LIN {X 0,Y 367.075,Z 1146.88,A -85,B 0,C 180,E1 14634.153,E2 14634.153} C_VEL
LIN {X 0,Y 373.267,Z 1130.589,A -85,B 0,C 180,E1 14631.284,E2 14631.284} C_VEL
LIN {X 0,Y 379.59,Z 1113.754,A -85,B 0,C 180,E1 14628.758,E2 14628.758} C_VEL
LIN {X 0,Y 386.074,Z 1095.539,A -85,B 0,C 180,E1 14626.458,E2 14626.458} C_VEL
LIN {X 0,Y 392.313,Z 1077.12,A -85,B 0,C 180,E1 14624.47,E2 14624.47} C_VEL
LIN {X 0,Y 398.602,Z 1056.8,A -85,B 0,C 180,E1 14622.633,E2 14622.633} C_VEL
LIN {X 0,Y 404.177,Z 1037.14,A -85,B 0,C 180,E1 14621.125,E2 14621.125} C_VEL
LIN {X 0,Y 409.615,Z 1015.322,A -85,B 0,C 180,E1 14619.744,E2 14619.744} C_VEL
LIN {X 0,Y 414.222,Z 994.195,A -85,B 0,C 180,E1 14618.639,E2 14618.639} C_VEL
LIN {X 0,Y 418.394,Z 971.046,A -85,B 0,C 180,E1 14617.677,E2 14617.677} C_VEL
LIN {X 0,Y 421.612,Z 949.02,A -85,B 0,C 180,E1 14616.963,E2 14616.963} C_VEL
LIN {X 0,Y 424.148,Z 924.511,A -85,B 0,C 180,E1 14616.384,E2 14616.384} C_VEL
LIN {X 0,Y 439.358,Z 688.452,A -85,B 0,C 180,E1 14612.27,E2 14612.27} C_VEL
LIN {X 0,Y 440.922,Z 663.001,A -85,B 0,C 180,E1 14611.82,E2 14611.82} C_VEL
LIN {X 0,Y 431.754,Z 648.158,A -85,B 0,C 180,E1 14609.595,E2 14609.595} C_VEL
LIN {X 0,Y 422.609,Z 634.496,A -85,B 0,C 180,E1 14607.17,E2 14607.17} C_VEL
LIN {X 0,Y 413.735,Z 622.138,A -85,B 0,C 180,E1 14604.562,E2 14604.562} C_VEL
LIN {X 0,Y 405.049,Z 611.055,A -85,B 0,C 180,E1 14601.695,E2 14601.695} C_VEL
LIN {X 0,Y 397.899,Z 602.317,A -85,B 0,C 180,E1 14598.991,E2 14598.991} C_VEL
LIN {X 0,Y 392.596,Z 596.37,A -85,B 0,C 180,E1 14596.726,E2 14596.726} C_VEL
LIN {X 0,Y 388.549,Z 591.744,A -85,B 0,C 180,E1 14594.76,E2 14594.76} C_VEL
LIN {X 0,Y 383.66,Z 586.476,A -85,B 0,C 180,E1 14592.034,E2 14592.034} C_VEL
LIN {X 0,Y 379.03,Z 581.897,A -85,B 0,C 180,E1 14588.878,E2 14588.878} C_VEL
LIN {X 0,Y 378.199,Z 580.649,A -85,B 0,C 180,E1 14587.749,E2 14587.749} C_VEL
LIN {X 0,Y 376.427,Z 578.063,A -85,B 0,C 180,E1 14582.131,E2 14582.131} C_VEL
LIN {X 0,Y 376.328,Z 577.802,A -85,B 0,C 180,E1 14578.477,E2 14578.477} C_VEL
LIN {X 0,Y 377.214,Z 579.561,A -85,B 0,C 180,E1 14573.608,E2 14573.608} C_VEL
LIN {X 0,Y 378.457,Z 581.248,A -85,B 0,C 180,E1 14570.879,E2 14570.879} C_VEL
LIN {X 0,Y 380.862,Z 586.157,A -85,B 0,C 180,E1 14566.488,E2 14566.488} C_VEL
LIN {X 0,Y 383.165,Z 591.028,A -85,B 0,C 180,E1 14563.318,E2 14563.318} C_VEL
LIN {X 0,Y 385.362,Z 595.637,A -85,B 0,C 180,E1 14560.809,E2 14560.809} C_VEL
LIN {X 0,Y 387.472,Z 600.181,A -85,B 0,C 180,E1 14558.663,E2 14558.663} C_VEL
LIN {X 0,Y 389.455,Z 603.852,A -85,B 0,C 180,E1 14557.19,E2 14557.19} C_VEL
LIN {X 0,Y 396.46,Z 614.138,A -85,B 0,C 180,E1 14554.01,E2 14554.01} C_VEL
LIN {X 0,Y 403.343,Z 624.564,A -85,B 0,C 180,E1 14551.335,E2 14551.335} C_VEL
LIN {X 0,Y 411.127,Z 636.839,A -85,B 0,C 180,E1 14548.677,E2 14548.677} C_VEL
LIN {X 0,Y 418.492,Z 649.282,A -85,B 0,C 180,E1 14546.419,E2 14546.419} C_VEL
LIN {X 0,Y 427.201,Z 664.773,A -85,B 0,C 180,E1 14544.001,E2 14544.001} C_VEL
LIN {X 0,Y 430.356,Z 671.029,A -85,B 0,C 180,E1 14543.17,E2 14543.17} C_VEL
LIN {X 0,Y 435.237,Z 722.791,A -85,B 0,C 180,E1 14540.824,E2 14540.824} C_VEL
LIN {X 0,Y 423.088,Z 947.316,A -85,B 0,C 180,E1 14537.248,E2 14537.248} C_VEL
LIN {X 0,Y 420.542,Z 970.15,A -85,B 0,C 180,E1 14536.723,E2 14536.723} C_VEL
LIN {X 0,Y 417.124,Z 991.912,A -85,B 0,C 180,E1 14536.04,E2 14536.04} C_VEL
LIN {X 0,Y 413.008,Z 1012.312,A -85,B 0,C 180,E1 14535.18,E2 14535.18} C_VEL
LIN {X 0,Y 407.851,Z 1033.865,A -85,B 0,C 180,E1 14534.028,E2 14534.028} C_VEL
LIN {X 0,Y 402.694,Z 1052.364,A -85,B 0,C 180,E1 14532.803,E2 14532.803} C_VEL
LIN {X 0,Y 396.609,Z 1071.682,A -85,B 0,C 180,E1 14531.242,E2 14531.242} C_VEL
LIN {X 0,Y 390.215,Z 1090.083,A -85,B 0,C 180,E1 14529.454,E2 14529.454} C_VEL
LIN {X 0,Y 383.57,Z 1107.397,A -85,B 0,C 180,E1 14527.399,E2 14527.399} C_VEL
LIN {X 0,Y 376.663,Z 1124.336,A -85,B 0,C 180,E1 14524.986,E2 14524.986} C_VEL
LIN {X 0,Y 370.434,Z 1138.925,A -85,B 0,C 180,E1 14522.488,E2 14522.488} C_VEL
LIN {X 0,Y 364.569,Z 1152.135,A -85,B 0,C 180,E1 14519.762,E2 14519.762} C_VEL
LIN {X 0,Y 359.259,Z 1164.199,A -85,B 0,C 180,E1 14516.799,E2 14516.799} C_VEL
LIN {X 0,Y 354.544,Z 1174.916,A -85,B 0,C 180,E1 14513.569,E2 14513.569} C_VEL
LIN {X 0,Y 350.568,Z 1184.53,A -85,B 0,C 180,E1 14510.014,E2 14510.014} C_VEL
LIN {X 0,Y 347.654,Z 1192.408,A -85,B 0,C 180,E1 14506.371,E2 14506.371} C_VEL
LIN {X 0,Y 345.722,Z 1198.398,A -85,B 0,C 180,E1 14502.697,E2 14502.697} C_VEL
LIN {X 0,Y 344.593,Z 1203.015,A -85,B 0,C 180,E1 14498.846,E2 14498.846} C_VEL
LIN {X 0,Y 344.142,Z 1205.734,A -85,B 0,C 180,E1 14495.335,E2 14495.335} C_VEL
LIN {X 0,Y 344.006,Z 1207.141,A -85,B 0,C 180,E1 14491.666,E2 14491.666} C_VEL
LIN {X 0,Y 344,Z 1207.177,A -85,B 0,C 180,E1 14488.501,E2 14488.501} C_VEL
LIN {X 0,Y 344.124,Z 1205.916,A -85,B 0,C 180,E1 14484.832,E2 14484.832} C_VEL
LIN {X 0,Y 344.544,Z 1203.27,A -85,B 0,C 180,E1 14481.321,E2 14481.321} C_VEL
LIN {X 0,Y 345.693,Z 1198.563,A -85,B 0,C 180,E1 14477.302,E2 14477.302} C_VEL
LIN {X 0,Y 347.601,Z 1192.614,A -85,B 0,C 180,E1 14473.627,E2 14473.627} C_VEL
LIN {X 0,Y 350.493,Z 1184.79,A -85,B 0,C 180,E1 14469.981,E2 14469.981} C_VEL
LIN {X 0,Y 354.698,Z 1174.638,A -85,B 0,C 180,E1 14466.228,E2 14466.228} C_VEL
LIN {X 0,Y 359.396,Z 1164.003,A -85,B 0,C 180,E1 14463.033,E2 14463.033} C_VEL
LIN {X 0,Y 364.916,Z 1151.502,A -85,B 0,C 180,E1 14459.981,E2 14459.981} C_VEL
LIN {X 0,Y 371.322,Z 1136.991,A -85,B 0,C 180,E1 14457.049,E2 14457.049} C_VEL
LIN {X 0,Y 377.667,Z 1122.208,A -85,B 0,C 180,E1 14454.564,E2 14454.564} C_VEL
LIN {X 0,Y 384.244,Z 1105.923,A -85,B 0,C 180,E1 14452.302,E2 14452.302} C_VEL
LIN {X 0,Y 390.941,Z 1088.307,A -85,B 0,C 180,E1 14450.254,E2 14450.254} C_VEL
LIN {X 0,Y 396.895,Z 1071.164,A -85,B 0,C 180,E1 14448.602,E2 14448.602} C_VEL
LIN {X 0,Y 400.054,Z 1061.338,A -85,B 0,C 180,E1 14447.776,E2 14447.776} C_VEL
LIN {X 0,Y 401.438,Z 1054.915,A -85,B 0,C 180,E1 14447.179,E2 14447.179} C_VEL
LIN {X 0,Y 401.841,Z 1038.851,A -85,B 0,C 180,E1 14445.454,E2 14445.454} C_VEL
LIN {X 0,Y 402.944,Z 1032.138,A -85,B 0,C 180,E1 14444.927,E2 14444.927} C_VEL
LIN {X 0,Y 408.068,Z 1010.972,A -85,B 0,C 180,E1 14443.814,E2 14443.814} C_VEL
LIN {X 0,Y 412.471,Z 989.311,A -85,B 0,C 180,E1 14442.921,E2 14442.921} C_VEL
LIN {X 0,Y 415.872,Z 967.674,A -85,B 0,C 180,E1 14442.264,E2 14442.264} C_VEL
LIN {X 0,Y 418.4,Z 943.81,A -85,B 0,C 180,E1 14441.739,E2 14441.739} C_VEL
LIN {X 0,Y 430.607,Z 723.448,A -85,B 0,C 180,E1 14438.192,E2 14438.192} C_VEL
LIN {X 0,Y 426.313,Z 675.47,A -85,B 0,C 180,E1 14435.982,E2 14435.982} C_VEL
LIN {X 0,Y 418.355,Z 660.566,A -85,B 0,C 180,E1 14433.758,E2 14433.758} C_VEL
LIN {X 0,Y 410.661,Z 647.161,A -85,B 0,C 180,E1 14431.403,E2 14431.403} C_VEL
LIN {X 0,Y 402.691,Z 634.171,A -85,B 0,C 180,E1 14428.675,E2 14428.675} C_VEL
LIN {X 0,Y 397.146,Z 625.543,A -85,B 0,C 180,E1 14426.544,E2 14426.544} C_VEL
LIN {X 0,Y 391.843,Z 617.436,A -85,B 0,C 180,E1 14424.257,E2 14424.257} C_VEL
LIN {X 0,Y 386.128,Z 608.96,A -85,B 0,C 180,E1 14421.415,E2 14421.415} C_VEL
LIN {X 0,Y 380.176,Z 600.315,A -85,B 0,C 180,E1 14417.764,E2 14417.764} C_VEL
LIN {X 0,Y 377.816,Z 595.977,A -85,B 0,C 180,E1 14415.346,E2 14415.346} C_VEL
LIN {X 0,Y 375.944,Z 591.854,A -85,B 0,C 180,E1 14412.441,E2 14412.441} C_VEL
LIN {X 0,Y 373.797,Z 587.386,A -85,B 0,C 180,E1 14407.996,E2 14407.996} C_VEL
LIN {X 0,Y 372.205,Z 585.048,A -85,B 0,C 180,E1 14402.463,E2 14402.463} C_VEL
LIN {X 0,Y 372.164,Z 584.871,A -85,B 0,C 180,E1 14398.922,E2 14398.922} C_VEL
LIN {X 0,Y 372.818,Z 585.725,A -85,B 0,C 180,E1 14396.617,E2 14396.617} C_VEL
LIN {X 0,Y 377.49,Z 589.328,A -85,B 0,C 180,E1 14391.777,E2 14391.777} C_VEL
LIN {X 0,Y 381.514,Z 593.671,A -85,B 0,C 180,E1 14388.817,E2 14388.817} C_VEL
LIN {X 0,Y 383.391,Z 595.508,A -85,B 0,C 180,E1 14387.651,E2 14387.651} C_VEL
LIN {X 0,Y 388.761,Z 601.407,A -85,B 0,C 180,E1 14384.714,E2 14384.714} C_VEL
LIN {X 0,Y 394.144,Z 607.712,A -85,B 0,C 180,E1 14382.2,E2 14382.2} C_VEL
LIN {X 0,Y 398.695,Z 613.148,A -85,B 0,C 180,E1 14380.325,E2 14380.325} C_VEL
LIN {X 0,Y 405.06,Z 621.01,A -85,B 0,C 180,E1 14377.962,E2 14377.962} C_VEL
LIN {X 0,Y 414.608,Z 633.741,A -85,B 0,C 180,E1 14374.846,E2 14374.846} C_VEL
LIN {X 0,Y 423.799,Z 647.185,A -85,B 0,C 180,E1 14372.189,E2 14372.189} C_VEL
LIN {X 0,Y 433.257,Z 662.083,A -85,B 0,C 180,E1 14369.717,E2 14369.717} C_VEL
LIN {X 0,Y 436.289,Z 667.482,A -85,B 0,C 180,E1 14368.959,E2 14368.959} C_VEL
LIN {X 0,Y 420.331,Z 909.767,A -85,B 0,C 180,E1 14364.754,E2 14364.754} C_VEL
LIN {X 0,Y 417.975,Z 937.62,A -85,B 0,C 180,E1 14364.195,E2 14364.195} C_VEL
LIN {X 0,Y 414.977,Z 961.048,A -85,B 0,C 180,E1 14363.542,E2 14363.542} C_VEL
LIN {X 0,Y 411.076,Z 983.796,A -85,B 0,C 180,E1 14362.689,E2 14362.689} C_VEL
LIN {X 0,Y 406.363,Z 1006.888,A -85,B 0,C 180,E1 14361.598,E2 14361.598} C_VEL
LIN {X 0,Y 400.948,Z 1028.836,A -85,B 0,C 180,E1 14360.293,E2 14360.293} C_VEL
LIN {X 0,Y 394.958,Z 1050.407,A -85,B 0,C 180,E1 14358.753,E2 14358.753} C_VEL
LIN {X 0,Y 388.718,Z 1070.338,A -85,B 0,C 180,E1 14357.027,E2 14357.027} C_VEL
LIN {X 0,Y 381.72,Z 1090.963,A -85,B 0,C 180,E1 14354.903,E2 14354.903} C_VEL
LIN {X 0,Y 375.382,Z 1108.288,A -85,B 0,C 180,E1 14352.782,E2 14352.782} C_VEL
LIN {X 0,Y 368.175,Z 1127.067,A -85,B 0,C 180,E1 14350.062,E2 14350.062} C_VEL
LIN {X 0,Y 362.387,Z 1141.642,A -85,B 0,C 180,E1 14347.572,E2 14347.572} C_VEL
LIN {X 0,Y 355.922,Z 1157.783,A -85,B 0,C 180,E1 14344.316,E2 14344.316} C_VEL
LIN {X 0,Y 350.848,Z 1170.642,A -85,B 0,C 180,E1 14341.242,E2 14341.242} C_VEL
LIN {X 0,Y 345.924,Z 1183.598,A -85,B 0,C 180,E1 14337.546,E2 14337.546} C_VEL
LIN {X 0,Y 342.26,Z 1194.124,A -85,B 0,C 180,E1 14333.958,E2 14333.958} C_VEL
LIN {X 0,Y 339.449,Z 1203.219,A -85,B 0,C 180,E1 14330.159,E2 14330.159} C_VEL
LIN {X 0,Y 337.719,Z 1210.045,A -85,B 0,C 180,E1 14326.689,E2 14326.689} C_VEL
LIN {X 0,Y 336.509,Z 1216.429,A -85,B 0,C 180,E1 14322.527,E2 14322.527} C_VEL
LIN {X 0,Y 336.076,Z 1220.328,A -85,B 0,C 180,E1 14319.072,E2 14319.072} C_VEL
LIN {X 0,Y 335.938,Z 1223.253,A -85,B 0,C 180,E1 14315.294,E2 14315.294} C_VEL
LIN {X 0,Y 335.967,Z 1224.501,A -85,B 0,C 180,E1 14311.705,E2 14311.705} C_VEL
LIN {X 0,Y 335.969,Z 1224.547,A -85,B 0,C 180,E1 14308.636,E2 14308.636} C_VEL
LIN {X 0,Y 335.949,Z 1223.537,A -85,B 0,C 180,E1 14305.391,E2 14305.391} C_VEL
LIN {X 0,Y 336.03,Z 1220.984,A -85,B 0,C 180,E1 14301.616,E2 14301.616} C_VEL
LIN {X 0,Y 336.414,Z 1217.058,A -85,B 0,C 180,E1 14297.992,E2 14297.992} C_VEL
LIN {X 0,Y 337.33,Z 1211.819,A -85,B 0,C 180,E1 14294.352,E2 14294.352} C_VEL
LIN {X 0,Y 339.139,Z 1204.281,A -85,B 0,C 180,E1 14290.361,E2 14290.361} C_VEL
LIN {X 0,Y 341.68,Z 1195.859,A -85,B 0,C 180,E1 14286.731,E2 14286.731} C_VEL
LIN {X 0,Y 345.337,Z 1185.139,A -85,B 0,C 180,E1 14282.963,E2 14282.963} C_VEL
LIN {X 0,Y 349.618,Z 1173.731,A -85,B 0,C 180,E1 14279.589,E2 14279.589} C_VEL
LIN {X 0,Y 355.013,Z 1159.928,A -85,B 0,C 180,E1 14276.188,E2 14276.188} C_VEL
LIN {X 0,Y 361.027,Z 1144.988,A -85,B 0,C 180,E1 14273.06,E2 14273.06} C_VEL
LIN {X 0,Y 367.396,Z 1128.826,A -85,B 0,C 180,E1 14270.242,E2 14270.242} C_VEL
LIN {X 0,Y 374.235,Z 1111.205,A -85,B 0,C 180,E1 14267.621,E2 14267.621} C_VEL
LIN {X 0,Y 380.574,Z 1093.875,A -85,B 0,C 180,E1 14265.455,E2 14265.455} C_VEL
LIN {X 0,Y 387.377,Z 1074.25,A -85,B 0,C 180,E1 14263.361,E2 14263.361} C_VEL
LIN {X 0,Y 393.417,Z 1055.087,A -85,B 0,C 180,E1 14261.652,E2 14261.652} C_VEL
LIN {X 0,Y 399.608,Z 1033.598,A -85,B 0,C 180,E1 14260.036,E2 14260.036} C_VEL
LIN {X 0,Y 404.692,Z 1013.376,A -85,B 0,C 180,E1 14258.786,E2 14258.786} C_VEL
LIN {X 0,Y 409.537,Z 991.477,A -85,B 0,C 180,E1 14257.662,E2 14257.662} C_VEL
LIN {X 0,Y 413.522,Z 969.319,A -85,B 0,C 180,E1 14256.767,E2 14256.767} C_VEL
LIN {X 0,Y 416.916,Z 946.2,A -85,B 0,C 180,E1 14256.036,E2 14256.036} C_VEL
LIN {X 0,Y 419.267,Z 922.548,A -85,B 0,C 180,E1 14255.498,E2 14255.498} C_VEL
LIN {X 0,Y 435.003,Z 684.514,A -85,B 0,C 180,E1 14251.344,E2 14251.344} C_VEL
LIN {X 0,Y 436.072,Z 666.851,A -85,B 0,C 180,E1 14251.02,E2 14251.02} C_VEL
LIN {X 0,Y 426.546,Z 651.468,A -85,B 0,C 180,E1 14248.607,E2 14248.607} C_VEL
LIN {X 0,Y 417.357,Z 637.74,A -85,B 0,C 180,E1 14246.042,E2 14246.042} C_VEL
LIN {X 0,Y 408.027,Z 624.866,A -85,B 0,C 180,E1 14243.123,E2 14243.123} C_VEL
LIN {X 0,Y 399.618,Z 614.248,A -85,B 0,C 180,E1 14240.123,E2 14240.123} C_VEL
LIN {X 0,Y 394.405,Z 608.036,A -85,B 0,C 180,E1 14238.017,E2 14238.017} C_VEL
LIN {X 0,Y 390.537,Z 603.573,A -85,B 0,C 180,E1 14236.281,E2 14236.281} C_VEL
LIN {X 0,Y 386.859,Z 599.291,A -85,B 0,C 180,E1 14234.443,E2 14234.443} C_VEL
LIN {X 0,Y 382.19,Z 594.174,A -85,B 0,C 180,E1 14231.775,E2 14231.775} C_VEL
LIN {X 0,Y 377.662,Z 589.568,A -85,B 0,C 180,E1 14228.603,E2 14228.603} C_VEL
LIN {X 0,Y 376.14,Z 588.195,A -85,B 0,C 180,E1 14227.331,E2 14227.331} C_VEL
LIN {X 0,Y 372.214,Z 584.956,A -85,B 0,C 180,E1 14222.617,E2 14222.617} C_VEL
LIN {X 0,Y 371.979,Z 584.446,A -85,B 0,C 180,E1 14218.922,E2 14218.922} C_VEL
LIN {X 0,Y 372.563,Z 585.871,A -85,B 0,C 180,E1 14214.456,E2 14214.456} C_VEL
LIN {X 0,Y 374.026,Z 587.938,A -85,B 0,C 180,E1 14210.925,E2 14210.925} C_VEL
LIN {X 0,Y 376.302,Z 592.669,A -85,B 0,C 180,E1 14206.634,E2 14206.634} C_VEL
LIN {X 0,Y 378.573,Z 597.575,A -85,B 0,C 180,E1 14203.426,E2 14203.426} C_VEL
LIN {X 0,Y 381.302,Z 602.118,A -85,B 0,C 180,E1 14201.183,E2 14201.183} C_VEL
LIN {X 0,Y 387.44,Z 610.898,A -85,B 0,C 180,E1 14197.665,E2 14197.665} C_VEL
LIN {X 0,Y 394.439,Z 621.431,A -85,B 0,C 180,E1 14194.392,E2 14194.392} C_VEL
LIN {X 0,Y 401.014,Z 631.624,A -85,B 0,C 180,E1 14191.763,E2 14191.763} C_VEL
LIN {X 0,Y 408.466,Z 643.595,A -85,B 0,C 180,E1 14189.147,E2 14189.147} C_VEL
LIN {X 0,Y 415.589,Z 655.893,A -85,B 0,C 180,E1 14186.896,E2 14186.896} C_VEL
LIN {X 0,Y 424.048,Z 671.21,A -85,B 0,C 180,E1 14184.483,E2 14184.483} C_VEL
LIN {X 0,Y 426.192,Z 675.798,A -85,B 0,C 180,E1 14183.892,E2 14183.892} C_VEL
LIN {X 0,Y 430.502,Z 724.672,A -85,B 0,C 180,E1 14181.658,E2 14181.658} C_VEL
LIN {X 0,Y 418.035,Z 946.95,A -85,B 0,C 180,E1 14178.099,E2 14178.099} C_VEL
LIN {X 0,Y 415.411,Z 969.946,A -85,B 0,C 180,E1 14177.569,E2 14177.569} C_VEL
LIN {X 0,Y 411.915,Z 991.659,A -85,B 0,C 180,E1 14176.888,E2 14176.888} C_VEL
LIN {X 0,Y 407.724,Z 1011.938,A -85,B 0,C 180,E1 14176.034,E2 14176.034} C_VEL
LIN {X 0,Y 402.43,Z 1033.542,A -85,B 0,C 180,E1 14174.879,E2 14174.879} C_VEL
LIN {X 0,Y 396.9,Z 1052.853,A -85,B 0,C 180,E1 14173.594,E2 14173.594} C_VEL
LIN {X 0,Y 390.622,Z 1072.154,A -85,B 0,C 180,E1 14172.017,E2 14172.017} C_VEL
LIN {X 0,Y 384.048,Z 1090.491,A -85,B 0,C 180,E1 14170.215,E2 14170.215} C_VEL
LIN {X 0,Y 377.207,Z 1107.761,A -85,B 0,C 180,E1 14168.142,E2 14168.142} C_VEL
LIN {X 0,Y 370.077,Z 1124.648,A -85,B 0,C 180,E1 14165.703,E2 14165.703} C_VEL
LIN {X 0,Y 363.639,Z 1139.221,A -85,B 0,C 180,E1 14163.173,E2 14163.173} C_VEL
LIN {X 0,Y 357.558,Z 1152.397,A -85,B 0,C 180,E1 14160.407,E2 14160.407} C_VEL
LIN {X 0,Y 352.035,Z 1164.44,A -85,B 0,C 180,E1 14157.395,E2 14157.395} C_VEL
LIN {X 0,Y 347.164,Z 1175.045,A -85,B 0,C 180,E1 14154.14,E2 14154.14} C_VEL
LIN {X 0,Y 342.954,Z 1184.754,A -85,B 0,C 180,E1 14150.478,E2 14150.478} C_VEL
LIN {X 0,Y 339.886,Z 1192.626,A -85,B 0,C 180,E1 14146.756,E2 14146.756} C_VEL
LIN {X 0,Y 337.843,Z 1198.611,A -85,B 0,C 180,E1 14142.998,E2 14142.998} C_VEL
LIN {X 0,Y 336.639,Z 1203.222,A -85,B 0,C 180,E1 14139.057,E2 14139.057} C_VEL
LIN {X 0,Y 336.156,Z 1205.941,A -85,B 0,C 180,E1 14135.462,E2 14135.462} C_VEL
LIN {X 0,Y 336.009,Z 1207.345,A -85,B 0,C 180,E1 14131.705,E2 14131.705} C_VEL
LIN {X 0,Y 336.003,Z 1207.381,A -85,B 0,C 180,E1 14128.465,E2 14128.465} C_VEL
LIN {X 0,Y 336.136,Z 1206.122,A -85,B 0,C 180,E1 14124.709,E2 14124.709} C_VEL
LIN {X 0,Y 336.585,Z 1203.476,A -85,B 0,C 180,E1 14121.114,E2 14121.114} C_VEL
LIN {X 0,Y 337.812,Z 1198.774,A -85,B 0,C 180,E1 14117,E2 14117} C_VEL
LIN {X 0,Y 339.833,Z 1192.827,A -85,B 0,C 180,E1 14113.242,E2 14113.242} C_VEL
LIN {X 0,Y 342.877,Z 1185.011,A -85,B 0,C 180,E1 14109.517,E2 14109.517} C_VEL
LIN {X 0,Y 347.064,Z 1175.368,A -85,B 0,C 180,E1 14105.853,E2 14105.853} C_VEL
LIN {X 0,Y 351.911,Z 1164.797,A -85,B 0,C 180,E1 14102.595,E2 14102.595} C_VEL
LIN {X 0,Y 357.418,Z 1152.841,A -85,B 0,C 180,E1 14099.58,E2 14099.58} C_VEL
LIN {X 0,Y 363.832,Z 1138.95,A -85,B 0,C 180,E1 14096.664,E2 14096.664} C_VEL
LIN {X 0,Y 370.307,Z 1124.322,A -85,B 0,C 180,E1 14094.132,E2 14094.132} C_VEL
LIN {X 0,Y 377.464,Z 1107.365,A -85,B 0,C 180,E1 14091.696,E2 14091.696} C_VEL
LIN {X 0,Y 384.333,Z 1090.037,A -85,B 0,C 180,E1 14089.625,E2 14089.625} C_VEL
LIN {X 0,Y 390.92,Z 1071.626,A -85,B 0,C 180,E1 14087.825,E2 14087.825} C_VEL
LIN {X 0,Y 397.623,Z 1050.801,A -85,B 0,C 180,E1 14086.151,E2 14086.151} C_VEL
LIN {X 0,Y 402.944,Z 1032.138,A -85,B 0,C 180,E1 14084.927,E2 14084.927} C_VEL
LIN {X 0,Y 404.109,Z 1025.327,A -85,B 0,C 180,E1 14084.422,E2 14084.422} C_VEL
LIN {X 0,Y 404.184,Z 1008.202,A -85,B 0,C 180,E1 14082.925,E2 14082.925} C_VEL
LIN {X 0,Y 405.005,Z 1001.057,A -85,B 0,C 180,E1 14082.517,E2 14082.517} C_VEL
LIN {X 0,Y 408.853,Z 980.543,A -85,B 0,C 180,E1 14081.772,E2 14081.772} C_VEL
LIN {X 0,Y 412.137,Z 957.278,A -85,B 0,C 180,E1 14081.151,E2 14081.151} C_VEL
LIN {X 0,Y 414.107,Z 934.287,A -85,B 0,C 180,E1 14080.702,E2 14080.702} C_VEL
LIN {X 0,Y 425.986,Z 725.009,A -85,B 0,C 180,E1 14077.335,E2 14077.335} C_VEL
LIN {X 0,Y 422.146,Z 679.945,A -85,B 0,C 180,E1 14075.223,E2 14075.223} C_VEL
LIN {X 0,Y 414.286,Z 665.02,A -85,B 0,C 180,E1 14072.932,E2 14072.932} C_VEL
LIN {X 0,Y 406.152,Z 650.7,A -85,B 0,C 180,E1 14070.31,E2 14070.31} C_VEL
LIN {X 0,Y 398.248,Z 637.719,A -85,B 0,C 180,E1 14067.434,E2 14067.434} C_VEL
LIN {X 0,Y 390.354,Z 625.349,A -85,B 0,C 180,E1 14064.074,E2 14064.074} C_VEL
LIN {X 0,Y 384.379,Z 616.349,A -85,B 0,C 180,E1 14061.038,E2 14061.038} C_VEL
LIN {X 0,Y 378.669,Z 607.88,A -85,B 0,C 180,E1 14057.44,E2 14057.44} C_VEL
LIN {X 0,Y 375.726,Z 603.557,A -85,B 0,C 180,E1 14055.118,E2 14055.118} C_VEL
LIN {X 0,Y 372.866,Z 599.149,A -85,B 0,C 180,E1 14052.231,E2 14052.231} C_VEL
LIN {X 0,Y 370.187,Z 594.511,A -85,B 0,C 180,E1 14047.918,E2 14047.918} C_VEL
LIN {X 0,Y 369.372,Z 592.509,A -85,B 0,C 180,E1 14042.327,E2 14042.327} C_VEL
LIN {X 0,Y 370.667,Z 592.831,A -85,B 0,C 180,E1 14038.454,E2 14038.454} C_VEL
LIN {X 0,Y 373.543,Z 595.181,A -85,B 0,C 180,E1 14034.47,E2 14034.47} C_VEL
LIN {X 0,Y 376.227,Z 597.128,A -85,B 0,C 180,E1 14031.979,E2 14031.979} C_VEL
LIN {X 0,Y 380.298,Z 601.548,A -85,B 0,C 180,E1 14028.934,E2 14028.934} C_VEL
LIN {X 0,Y 382.028,Z 603.36,A -85,B 0,C 180,E1 14027.837,E2 14027.837} C_VEL
LIN {X 0,Y 387.191,Z 609.12,A -85,B 0,C 180,E1 14024.958,E2 14024.958} C_VEL
LIN {X 0,Y 392.341,Z 615.24,A -85,B 0,C 180,E1 14022.499,E2 14022.499} C_VEL
LIN {X 0,Y 398.203,Z 622.289,A -85,B 0,C 180,E1 14020.07,E2 14020.07} C_VEL
LIN {X 0,Y 406.204,Z 632.737,A -85,B 0,C 180,E1 14017.151,E2 14017.151} C_VEL
LIN {X 0,Y 415.104,Z 645.203,A -85,B 0,C 180,E1 14014.305,E2 14014.305} C_VEL
LIN {X 0,Y 424.045,Z 658.849,A -85,B 0,C 180,E1 14011.747,E2 14011.747} C_VEL
LIN {X 0,Y 431.56,Z 671.215,A -85,B 0,C 180,E1 14009.775,E2 14009.775} C_VEL
LIN {X 0,Y 415.043,Z 915.504,A -85,B 0,C 180,E1 14005.522,E2 14005.522} C_VEL
LIN {X 0,Y 412.777,Z 939.766,A -85,B 0,C 180,E1 14005.01,E2 14005.01} C_VEL
LIN {X 0,Y 409.536,Z 963.776,A -85,B 0,C 180,E1 14004.32,E2 14004.32} C_VEL
LIN {X 0,Y 405.599,Z 985.702,A -85,B 0,C 180,E1 14003.479,E2 14003.479} C_VEL
LIN {X 0,Y 400.746,Z 1008.459,A -85,B 0,C 180,E1 14002.381,E2 14002.381} C_VEL
LIN {X 0,Y 395.486,Z 1029.168,A -85,B 0,C 180,E1 14001.14,E2 14001.14} C_VEL
LIN {X 0,Y 389.325,Z 1050.692,A -85,B 0,C 180,E1 13999.593,E2 13999.593} C_VEL
LIN {X 0,Y 382.921,Z 1070.532,A -85,B 0,C 180,E1 13997.864,E2 13997.864} C_VEL
LIN {X 0,Y 375.678,Z 1091.182,A -85,B 0,C 180,E1 13995.72,E2 13995.72} C_VEL
LIN {X 0,Y 369.079,Z 1108.619,A -85,B 0,C 180,E1 13993.561,E2 13993.561} C_VEL
LIN {X 0,Y 361.473,Z 1127.69,A -85,B 0,C 180,E1 13990.752,E2 13990.752} C_VEL
LIN {X 0,Y 355.134,Z 1143.073,A -85,B 0,C 180,E1 13988.067,E2 13988.067} C_VEL
LIN {X 0,Y 348.789,Z 1158.21,A -85,B 0,C 180,E1 13984.926,E2 13984.926} C_VEL
LIN {X 0,Y 343.511,Z 1171.033,A -85,B 0,C 180,E1 13981.792,E2 13981.792} C_VEL
LIN {X 0,Y 338.583,Z 1183.352,A -85,B 0,C 180,E1 13978.196,E2 13978.196} C_VEL
LIN {X 0,Y 334.875,Z 1193.407,A -85,B 0,C 180,E1 13974.709,E2 13974.709} C_VEL
LIN {X 0,Y 331.724,Z 1202.993,A -85,B 0,C 180,E1 13970.65,E2 13970.65} C_VEL
LIN {X 0,Y 329.872,Z 1209.824,A -85,B 0,C 180,E1 13967.098,E2 13967.098} C_VEL
LIN {X 0,Y 328.569,Z 1216.217,A -85,B 0,C 180,E1 13962.835,E2 13962.835} C_VEL
LIN {X 0,Y 328.089,Z 1220.118,A -85,B 0,C 180,E1 13959.295,E2 13959.295} C_VEL
LIN {X 0,Y 327.941,Z 1223.047,A -85,B 0,C 180,E1 13955.423,E2 13955.423} C_VEL
LIN {X 0,Y 327.969,Z 1224.297,A -85,B 0,C 180,E1 13951.747,E2 13951.747} C_VEL
LIN {X 0,Y 327.972,Z 1224.342,A -85,B 0,C 180,E1 13948.602,E2 13948.602} C_VEL
LIN {X 0,Y 327.947,Z 1223.331,A -85,B 0,C 180,E1 13945.278,E2 13945.278} C_VEL
LIN {X 0,Y 328.049,Z 1220.773,A -85,B 0,C 180,E1 13941.411,E2 13941.411} C_VEL
LIN {X 0,Y 328.462,Z 1216.845,A -85,B 0,C 180,E1 13937.697,E2 13937.697} C_VEL
LIN {X 0,Y 329.523,Z 1211.334,A -85,B 0,C 180,E1 13933.79,E2 13933.79} C_VEL
LIN {X 0,Y 331.48,Z 1203.753,A -85,B 0,C 180,E1 13929.738,E2 13929.738} C_VEL
LIN {X 0,Y 334.395,Z 1194.772,A -85,B 0,C 180,E1 13925.818,E2 13925.818} C_VEL
LIN {X 0,Y 338.187,Z 1184.302,A -85,B 0,C 180,E1 13922.133,E2 13922.133} C_VEL
LIN {X 0,Y 342.991,Z 1172.258,A -85,B 0,C 180,E1 13918.547,E2 13918.547} C_VEL
LIN {X 0,Y 348.56,Z 1158.62,A -85,B 0,C 180,E1 13915.191,E2 13915.191} C_VEL
LIN {X 0,Y 354.768,Z 1143.811,A -85,B 0,C 180,E1 13912.092,E2 13912.092} C_VEL
LIN {X 0,Y 361.265,Z 1128.002,A -85,B 0,C 180,E1 13909.32,E2 13909.32} C_VEL
LIN {X 0,Y 368.465,Z 1110.005,A -85,B 0,C 180,E1 13906.644,E2 13906.644} C_VEL
LIN {X 0,Y 374.959,Z 1092.839,A -85,B 0,C 180,E1 13904.495,E2 13904.495} C_VEL
LIN {X 0,Y 382.157,Z 1072.52,A -85,B 0,C 180,E1 13902.344,E2 13902.344} C_VEL
LIN {X 0,Y 388.351,Z 1053.384,A -85,B 0,C 180,E1 13900.648,E2 13900.648} C_VEL
LIN {X 0,Y 394.913,Z 1030.858,A -85,B 0,C 180,E1 13898.988,E2 13898.988} C_VEL
LIN {X 0,Y 400.273,Z 1009.852,A -85,B 0,C 180,E1 13897.714,E2 13897.714} C_VEL
LIN {X 0,Y 405.282,Z 986.662,A -85,B 0,C 180,E1 13896.58,E2 13896.58} C_VEL
LIN {X 0,Y 409.25,Z 964.66,A -85,B 0,C 180,E1 13895.728,E2 13895.728} C_VEL
LIN {X 0,Y 412.577,Z 940.316,A -85,B 0,C 180,E1 13895.019,E2 13895.019} C_VEL
LIN {X 0,Y 414.858,Z 916.144,A -85,B 0,C 180,E1 13894.505,E2 13894.505} C_VEL
LIN {X 0,Y 431.263,Z 673.298,A -85,B 0,C 180,E1 13890.275,E2 13890.275} C_VEL
LIN {X 0,Y 431.29,Z 670.84,A -85,B 0,C 180,E1 13890.205,E2 13890.205} C_VEL
LIN {X 0,Y 422.219,Z 656.099,A -85,B 0,C 180,E1 13887.809,E2 13887.809} C_VEL
LIN {X 0,Y 414.094,Z 643.876,A -85,B 0,C 180,E1 13885.455,E2 13885.455} C_VEL
LIN {X 0,Y 405.546,Z 631.859,A -85,B 0,C 180,E1 13882.697,E2 13882.697} C_VEL
LIN {X 0,Y 397.558,Z 621.582,A -85,B 0,C 180,E1 13879.772,E2 13879.772} C_VEL
LIN {X 0,Y 392.439,Z 615.373,A -85,B 0,C 180,E1 13877.65,E2 13877.65} C_VEL
LIN {X 0,Y 388.212,Z 610.438,A -85,B 0,C 180,E1 13875.691,E2 13875.691} C_VEL
LIN {X 0,Y 385.182,Z 606.839,A -85,B 0,C 180,E1 13874.124,E2 13874.124} C_VEL
LIN {X 0,Y 380.729,Z 601.873,A -85,B 0,C 180,E1 13871.513,E2 13871.513} C_VEL
LIN {X 0,Y 376.216,Z 597.104,A -85,B 0,C 180,E1 13868.252,E2 13868.252} C_VEL
LIN {X 0,Y 370.891,Z 592.812,A -85,B 0,C 180,E1 13862.472,E2 13862.472} C_VEL
LIN {X 0,Y 369.23,Z 592.013,A -85,B 0,C 180,E1 13858.603,E2 13858.603} C_VEL
LIN {X 0,Y 369.278,Z 593.43,A -85,B 0,C 180,E1 13853.626,E2 13853.626} C_VEL
LIN {X 0,Y 370.256,Z 594.856,A -85,B 0,C 180,E1 13851.145,E2 13851.145} C_VEL
LIN {X 0,Y 373.376,Z 600.109,A -85,B 0,C 180,E1 13846.764,E2 13846.764} C_VEL
LIN {X 0,Y 376.895,Z 605.384,A -85,B 0,C 180,E1 13843.588,E2 13843.588} C_VEL
LIN {X 0,Y 379.887,Z 609.878,A -85,B 0,C 180,E1 13841.429,E2 13841.429} C_VEL
LIN {X 0,Y 385.584,Z 618.181,A -85,B 0,C 180,E1 13838.073,E2 13838.073} C_VEL
LIN {X 0,Y 392.353,Z 628.597,A -85,B 0,C 180,E1 13834.812,E2 13834.812} C_VEL
LIN {X 0,Y 398.708,Z 638.682,A -85,B 0,C 180,E1 13832.195,E2 13832.195} C_VEL
LIN {X 0,Y 405.929,Z 650.509,A -85,B 0,C 180,E1 13829.589,E2 13829.589} C_VEL
LIN {X 0,Y 413.027,Z 663.055,A -85,B 0,C 180,E1 13827.285,E2 13827.285} C_VEL
LIN {X 0,Y 421.144,Z 678.064,A -85,B 0,C 180,E1 13824.91,E2 13824.91} C_VEL
LIN {X 0,Y 422.075,Z 680.407,A -85,B 0,C 180,E1 13824.635,E2 13824.635} C_VEL
LIN {X 0,Y 425.867,Z 726.268,A -85,B 0,C 180,E1 13822.516,E2 13822.516} C_VEL
LIN {X 0,Y 413.066,Z 946.695,A -85,B 0,C 180,E1 13818.968,E2 13818.968} C_VEL
LIN {X 0,Y 410.393,Z 969.603,A -85,B 0,C 180,E1 13818.44,E2 13818.44} C_VEL
LIN {X 0,Y 406.834,Z 991.242,A -85,B 0,C 180,E1 13817.764,E2 13817.764} C_VEL
LIN {X 0,Y 402.533,Z 1011.564,A -85,B 0,C 180,E1 13816.909,E2 13816.909} C_VEL
LIN {X 0,Y 397.128,Z 1033.12,A -85,B 0,C 180,E1 13815.759,E2 13815.759} C_VEL
LIN {X 0,Y 391.57,Z 1052.055,A -85,B 0,C 180,E1 13814.501,E2 13814.501} C_VEL
LIN {X 0,Y 384.964,Z 1071.9,A -85,B 0,C 180,E1 13812.882,E2 13812.882} C_VEL
LIN {X 0,Y 378.196,Z 1090.274,A -85,B 0,C 180,E1 13811.069,E2 13811.069} C_VEL
LIN {X 0,Y 371.135,Z 1107.572,A -85,B 0,C 180,E1 13808.981,E2 13808.981} C_VEL
LIN {X 0,Y 363.552,Z 1124.958,A -85,B 0,C 180,E1 13806.445,E2 13806.445} C_VEL
LIN {X 0,Y 356.897,Z 1139.516,A -85,B 0,C 180,E1 13803.883,E2 13803.883} C_VEL
LIN {X 0,Y 350.596,Z 1152.662,A -85,B 0,C 180,E1 13801.077,E2 13801.077} C_VEL
LIN {X 0,Y 344.85,Z 1164.681,A -85,B 0,C 180,E1 13798.015,E2 13798.015} C_VEL
LIN {X 0,Y 339.773,Z 1175.281,A -85,B 0,C 180,E1 13794.7,E2 13794.7} C_VEL
LIN {X 0,Y 335.365,Z 1184.975,A -85,B 0,C 180,E1 13790.963,E2 13790.963} C_VEL
LIN {X 0,Y 332.135,Z 1192.843,A -85,B 0,C 180,E1 13787.159,E2 13787.159} C_VEL
LIN {X 0,Y 329.972,Z 1198.824,A -85,B 0,C 180,E1 13783.314,E2 13783.314} C_VEL
LIN {X 0,Y 328.651,Z 1203.581,A -85,B 0,C 180,E1 13779.102,E2 13779.102} C_VEL
LIN {X 0,Y 328.156,Z 1206.255,A -85,B 0,C 180,E1 13775.42,E2 13775.42} C_VEL
LIN {X 0,Y 328.008,Z 1207.571,A -85,B 0,C 180,E1 13771.572,E2 13771.572} C_VEL
LIN {X 0,Y 328.009,Z 1207.564,A -85,B 0,C 180,E1 13768.253,E2 13768.253} C_VEL
LIN {X 0,Y 328.163,Z 1206.22,A -85,B 0,C 180,E1 13764.405,E2 13764.405} C_VEL
LIN {X 0,Y 328.672,Z 1203.531,A -85,B 0,C 180,E1 13760.722,E2 13760.722} C_VEL
LIN {X 0,Y 329.985,Z 1198.831,A -85,B 0,C 180,E1 13756.574,E2 13756.574} C_VEL
LIN {X 0,Y 332.202,Z 1192.734,A -85,B 0,C 180,E1 13752.664,E2 13752.664} C_VEL
LIN {X 0,Y 335.46,Z 1184.843,A -85,B 0,C 180,E1 13748.86,E2 13748.86} C_VEL
LIN {X 0,Y 339.898,Z 1175.104,A -85,B 0,C 180,E1 13745.124,E2 13745.124} C_VEL
LIN {X 0,Y 345.154,Z 1164.181,A -85,B 0,C 180,E1 13741.724,E2 13741.724} C_VEL
LIN {X 0,Y 351.115,Z 1151.736,A -85,B 0,C 180,E1 13738.593,E2 13738.593} C_VEL
LIN {X 0,Y 357.854,Z 1137.567,A -85,B 0,C 180,E1 13735.64,E2 13735.64} C_VEL
LIN {X 0,Y 364.635,Z 1122.816,A -85,B 0,C 180,E1 13733.093,E2 13733.093} C_VEL
LIN {X 0,Y 371.635,Z 1106.627,A -85,B 0,C 180,E1 13730.784,E2 13730.784} C_VEL
LIN {X 0,Y 378.734,Z 1089.145,A -85,B 0,C 180,E1 13728.7,E2 13728.7} C_VEL
LIN {X 0,Y 385.278,Z 1071.363,A -85,B 0,C 180,E1 13726.959,E2 13726.959} C_VEL
LIN {X 0,Y 392.172,Z 1050.49,A -85,B 0,C 180,E1 13725.278,E2 13725.278} C_VEL
LIN {X 0,Y 398.02,Z 1030.459,A -85,B 0,C 180,E1 13723.97,E2 13723.97} C_VEL
LIN {X 0,Y 403.189,Z 1009.3,A -85,B 0,C 180,E1 13722.878,E2 13722.878} C_VEL
LIN {X 0,Y 405.005,Z 1001.057,A -85,B 0,C 180,E1 13722.517,E2 13722.517} C_VEL
LIN {X 0,Y 405.864,Z 993.83,A -85,B 0,C 180,E1 13722.128,E2 13722.128} C_VEL
LIN {X 0,Y 405.302,Z 975.844,A -85,B 0,C 180,E1 13720.855,E2 13720.855} C_VEL
LIN {X 0,Y 405.743,Z 968.452,A -85,B 0,C 180,E1 13720.54,E2 13720.54} C_VEL
LIN {X 0,Y 408.494,Z 944.539,A -85,B 0,C 180,E1 13720,E2 13720} C_VEL
LIN {X 0,Y 421.47,Z 726.499,A -85,B 0,C 180,E1 13716.456,E2 13716.456} C_VEL
LIN {X 0,Y 418.115,Z 684.499,A -85,B 0,C 180,E1 13714.463,E2 13714.463} C_VEL
LIN {X 0,Y 410.491,Z 670.024,A -85,B 0,C 180,E1 13712.157,E2 13712.157} C_VEL
LIN {X 0,Y 403.355,Z 657.146,A -85,B 0,C 180,E1 13709.763,E2 13709.763} C_VEL
LIN {X 0,Y 395.816,Z 644.487,A -85,B 0,C 180,E1 13706.924,E2 13706.924} C_VEL
LIN {X 0,Y 388.115,Z 632.207,A -85,B 0,C 180,E1 13703.536,E2 13703.536} C_VEL
LIN {X 0,Y 382.646,Z 623.737,A -85,B 0,C 180,E1 13700.657,E2 13700.657} C_VEL
LIN {X 0,Y 377.096,Z 615.308,A -85,B 0,C 180,E1 13697.038,E2 13697.038} C_VEL
LIN {X 0,Y 374.422,Z 611.266,A -85,B 0,C 180,E1 13694.855,E2 13694.855} C_VEL
LIN {X 0,Y 371.645,Z 606.896,A -85,B 0,C 180,E1 13691.956,E2 13691.956} C_VEL
LIN {X 0,Y 369.16,Z 602.405,A -85,B 0,C 180,E1 13687.783,E2 13687.783} C_VEL
LIN {X 0,Y 368.388,Z 600.452,A -85,B 0,C 180,E1 13682.333,E2 13682.333} C_VEL
LIN {X 0,Y 369.602,Z 600.727,A -85,B 0,C 180,E1 13678.605,E2 13678.605} C_VEL
LIN {X 0,Y 372.277,Z 602.941,A -85,B 0,C 180,E1 13674.76,E2 13674.76} C_VEL
LIN {X 0,Y 374.968,Z 604.928,A -85,B 0,C 180,E1 13672.184,E2 13672.184} C_VEL
LIN {X 0,Y 379.085,Z 609.424,A -85,B 0,C 180,E1 13669.052,E2 13669.052} C_VEL
LIN {X 0,Y 380.785,Z 611.364,A -85,B 0,C 180,E1 13667.95,E2 13667.95} C_VEL
LIN {X 0,Y 385.496,Z 616.644,A -85,B 0,C 180,E1 13665.274,E2 13665.274} C_VEL
LIN {X 0,Y 390.554,Z 622.768,A -85,B 0,C 180,E1 13662.8,E2 13662.8} C_VEL
LIN {X 0,Y 396.754,Z 630.345,A -85,B 0,C 180,E1 13660.186,E2 13660.186} C_VEL
LIN {X 0,Y 404.773,Z 641.218,A -85,B 0,C 180,E1 13657.219,E2 13657.219} C_VEL
LIN {X 0,Y 412.604,Z 652.4,A -85,B 0,C 180,E1 13654.672,E2 13654.672} C_VEL
LIN {X 0,Y 421.066,Z 665.547,A -85,B 0,C 180,E1 13652.185,E2 13652.185} C_VEL
LIN {X 0,Y 426.88,Z 675.44,A -85,B 0,C 180,E1 13650.599,E2 13650.599} C_VEL
LIN {X 0,Y 410.015,Z 918.138,A -85,B 0,C 180,E1 13646.361,E2 13646.361} C_VEL
LIN {X 0,Y 407.731,Z 941.324,A -85,B 0,C 180,E1 13645.862,E2 13645.862} C_VEL
LIN {X 0,Y 404.182,Z 966.219,A -85,B 0,C 180,E1 13645.125,E2 13645.125} C_VEL
LIN {X 0,Y 400.201,Z 987.615,A -85,B 0,C 180,E1 13644.289,E2 13644.289} C_VEL
LIN {X 0,Y 394.949,Z 1011.051,A -85,B 0,C 180,E1 13643.129,E2 13643.129} C_VEL
LIN {X 0,Y 389.639,Z 1031.232,A -85,B 0,C 180,E1 13641.897,E2 13641.897} C_VEL
LIN {X 0,Y 382.802,Z 1053.958,A -85,B 0,C 180,E1 13640.212,E2 13640.212} C_VEL
LIN {X 0,Y 376.425,Z 1073.04,A -85,B 0,C 180,E1 13638.508,E2 13638.508} C_VEL
LIN {X 0,Y 368.998,Z 1093.267,A -85,B 0,C 180,E1 13636.342,E2 13636.342} C_VEL
LIN {X 0,Y 362.07,Z 1110.95,A -85,B 0,C 180,E1 13634.099,E2 13634.099} C_VEL
LIN {X 0,Y 354.714,Z 1128.579,A -85,B 0,C 180,E1 13631.425,E2 13631.425} C_VEL
LIN {X 0,Y 347.903,Z 1144.519,A -85,B 0,C 180,E1 13628.579,E2 13628.579} C_VEL
LIN {X 0,Y 341.462,Z 1159.175,A -85,B 0,C 180,E1 13625.435,E2 13625.435} C_VEL
LIN {X 0,Y 335.674,Z 1172.708,A -85,B 0,C 180,E1 13622.019,E2 13622.019} C_VEL
LIN {X 0,Y 330.643,Z 1184.714,A -85,B 0,C 180,E1 13618.344,E2 13618.344} C_VEL
LIN {X 0,Y 326.54,Z 1195.45,A -85,B 0,C 180,E1 13614.416,E2 13614.416} C_VEL
LIN {X 0,Y 323.656,Z 1203.924,A -85,B 0,C 180,E1 13610.597,E2 13610.597} C_VEL
LIN {X 0,Y 321.597,Z 1211.419,A -85,B 0,C 180,E1 13606.435,E2 13606.435} C_VEL
LIN {X 0,Y 320.517,Z 1216.659,A -85,B 0,C 180,E1 13602.613,E2 13602.613} C_VEL
LIN {X 0,Y 320.064,Z 1220.585,A -85,B 0,C 180,E1 13598.805,E2 13598.805} C_VEL
LIN {X 0,Y 319.945,Z 1223.135,A -85,B 0,C 180,E1 13594.84,E2 13594.84} C_VEL
LIN {X 0,Y 319.974,Z 1224.141,A -85,B 0,C 180,E1 13591.432,E2 13591.432} C_VEL
LIN {X 0,Y 319.971,Z 1224.089,A -85,B 0,C 180,E1 13588.209,E2 13588.209} C_VEL
LIN {X 0,Y 319.952,Z 1222.723,A -85,B 0,C 180,E1 13584.261,E2 13584.261} C_VEL
LIN {X 0,Y 320.107,Z 1219.887,A -85,B 0,C 180,E1 13580.471,E2 13580.471} C_VEL
LIN {X 0,Y 320.634,Z 1215.977,A -85,B 0,C 180,E1 13576.842,E2 13576.842} C_VEL
LIN {X 0,Y 322.077,Z 1209.401,A -85,B 0,C 180,E1 13572.38,E2 13572.38} C_VEL
LIN {X 0,Y 324.143,Z 1202.347,A -85,B 0,C 180,E1 13568.655,E2 13568.655} C_VEL
LIN {X 0,Y 327.546,Z 1192.628,A -85,B 0,C 180,E1 13564.506,E2 13564.506} C_VEL
LIN {X 0,Y 331.375,Z 1182.811,A -85,B 0,C 180,E1 13561.051,E2 13561.051} C_VEL
LIN {X 0,Y 337.011,Z 1169.358,A -85,B 0,C 180,E1 13557.117,E2 13557.117} C_VEL
LIN {X 0,Y 342.732,Z 1156.17,A -85,B 0,C 180,E1 13553.893,E2 13553.893} C_VEL
LIN {X 0,Y 349.36,Z 1140.887,A -85,B 0,C 180,E1 13550.766,E2 13550.766} C_VEL
LIN {X 0,Y 356.244,Z 1124.835,A -85,B 0,C 180,E1 13547.98,E2 13547.98} C_VEL
LIN {X 0,Y 363.604,Z 1106.779,A -85,B 0,C 180,E1 13545.365,E2 13545.365} C_VEL
LIN {X 0,Y 370.909,Z 1088.041,A -85,B 0,C 180,E1 13543.069,E2 13543.069} C_VEL
LIN {X 0,Y 377.938,Z 1068.277,A -85,B 0,C 180,E1 13541.063,E2 13541.063} C_VEL
LIN {X 0,Y 384.841,Z 1047.174,A -85,B 0,C 180,E1 13539.264,E2 13539.264} C_VEL
LIN {X 0,Y 390.651,Z 1027.106,A -85,B 0,C 180,E1 13537.852,E2 13537.852} C_VEL
LIN {X 0,Y 396.396,Z 1004.492,A -85,B 0,C 180,E1 13536.534,E2 13536.534} C_VEL
LIN {X 0,Y 401.016,Z 982.766,A -85,B 0,C 180,E1 13535.518,E2 13535.518} C_VEL
LIN {X 0,Y 405.44,Z 957.124,A -85,B 0,C 180,E1 13534.592,E2 13534.592} C_VEL
LIN {X 0,Y 408.431,Z 934.062,A -85,B 0,C 180,E1 13533.976,E2 13533.976} C_VEL
LIN {X 0,Y 411.309,Z 897.214,A -85,B 0,C 180,E1 13533.28,E2 13533.28} C_VEL
LIN {X 0,Y 426.731,Z 675.089,A -85,B 0,C 180,E1 13529.406,E2 13529.406} C_VEL
LIN {X 0,Y 417.862,Z 660.597,A -85,B 0,C 180,E1 13526.965,E2 13526.965} C_VEL
LIN {X 0,Y 409.176,Z 647.399,A -85,B 0,C 180,E1 13524.315,E2 13524.315} C_VEL
LIN {X 0,Y 399.972,Z 634.617,A -85,B 0,C 180,E1 13521.138,E2 13521.138} C_VEL
LIN {X 0,Y 392.23,Z 624.703,A -85,B 0,C 180,E1 13518.041,E2 13518.041} C_VEL
LIN {X 0,Y 386.918,Z 618.452,A -85,B 0,C 180,E1 13515.591,E2 13515.591} C_VEL
LIN {X 0,Y 383.516,Z 614.384,A -85,B 0,C 180,E1 13513.801,E2 13513.801} C_VEL
LIN {X 0,Y 379.275,Z 609.571,A -85,B 0,C 180,E1 13511.25,E2 13511.25} C_VEL
LIN {X 0,Y 374.868,Z 604.775,A -85,B 0,C 180,E1 13507.973,E2 13507.973} C_VEL
LIN {X 0,Y 369.718,Z 600.643,A -85,B 0,C 180,E1 13502.17,E2 13502.17} C_VEL
LIN {X 0,Y 368.176,Z 599.978,A -85,B 0,C 180,E1 13498.288,E2 13498.288} C_VEL
LIN {X 0,Y 368.396,Z 601.537,A -85,B 0,C 180,E1 13493.298,E2 13493.298} C_VEL
LIN {X 0,Y 369.204,Z 602.764,A -85,B 0,C 180,E1 13491.277,E2 13491.277} C_VEL
LIN {X 0,Y 372.191,Z 607.952,A -85,B 0,C 180,E1 13486.958,E2 13486.958} C_VEL
LIN {X 0,Y 375.556,Z 613.098,A -85,B 0,C 180,E1 13483.846,E2 13483.846} C_VEL
LIN {X 0,Y 378.48,Z 617.633,A -85,B 0,C 180,E1 13481.676,E2 13481.676} C_VEL
LIN {X 0,Y 383.812,Z 625.582,A -85,B 0,C 180,E1 13478.449,E2 13478.449} C_VEL
LIN {X 0,Y 390.363,Z 635.888,A -85,B 0,C 180,E1 13475.201,E2 13475.201} C_VEL
LIN {X 0,Y 396.426,Z 645.737,A -85,B 0,C 180,E1 13472.633,E2 13472.633} C_VEL
LIN {X 0,Y 403.412,Z 657.422,A -85,B 0,C 180,E1 13470.037,E2 13470.037} C_VEL
LIN {X 0,Y 411.375,Z 671.732,A -85,B 0,C 180,E1 13467.406,E2 13467.406} C_VEL
LIN {X 0,Y 417.996,Z 684.676,A -85,B 0,C 180,E1 13465.411,E2 13465.411} C_VEL
LIN {X 0,Y 421.333,Z 727.795,A -85,B 0,C 180,E1 13463.395,E2 13463.395} C_VEL
LIN {X 0,Y 408.194,Z 946.443,A -85,B 0,C 180,E1 13459.859,E2 13459.859} C_VEL
LIN {X 0,Y 405.452,Z 969.389,A -85,B 0,C 180,E1 13459.328,E2 13459.328} C_VEL
LIN {X 0,Y 401.737,Z 991.367,A -85,B 0,C 180,E1 13458.64,E2 13458.64} C_VEL
LIN {X 0,Y 397.144,Z 1012.469,A -85,B 0,C 180,E1 13457.747,E2 13457.747} C_VEL
LIN {X 0,Y 391.291,Z 1034.891,A -85,B 0,C 180,E1 13456.527,E2 13456.527} C_VEL
LIN {X 0,Y 385.368,Z 1054.428,A -85,B 0,C 180,E1 13455.203,E2 13455.203} C_VEL
LIN {X 0,Y 378.869,Z 1073.095,A -85,B 0,C 180,E1 13453.639,E2 13453.639} C_VEL
LIN {X 0,Y 371.926,Z 1091.266,A -85,B 0,C 180,E1 13451.813,E2 13451.813} C_VEL
LIN {X 0,Y 364.914,Z 1107.93,A -85,B 0,C 180,E1 13449.776,E2 13449.776} C_VEL
LIN {X 0,Y 357.091,Z 1125.264,A -85,B 0,C 180,E1 13447.214,E2 13447.214} C_VEL
LIN {X 0,Y 350.211,Z 1139.807,A -85,B 0,C 180,E1 13444.621,E2 13444.621} C_VEL
LIN {X 0,Y 343.685,Z 1152.924,A -85,B 0,C 180,E1 13441.774,E2 13441.774} C_VEL
LIN {X 0,Y 337.707,Z 1164.923,A -85,B 0,C 180,E1 13438.662,E2 13438.662} C_VEL
LIN {X 0,Y 332.416,Z 1175.518,A -85,B 0,C 180,E1 13435.285,E2 13435.285} C_VEL
LIN {X 0,Y 327.799,Z 1185.197,A -85,B 0,C 180,E1 13431.471,E2 13431.471} C_VEL
LIN {X 0,Y 324.401,Z 1193.058,A -85,B 0,C 180,E1 13427.581,E2 13427.581} C_VEL
LIN {X 0,Y 322.11,Z 1199.035,A -85,B 0,C 180,E1 13423.645,E2 13423.645} C_VEL
LIN {X 0,Y 320.705,Z 1203.788,A -85,B 0,C 180,E1 13419.33,E2 13419.33} C_VEL
LIN {X 0,Y 320.171,Z 1206.461,A -85,B 0,C 180,E1 13415.555,E2 13415.555} C_VEL
LIN {X 0,Y 320.012,Z 1207.775,A -85,B 0,C 180,E1 13411.611,E2 13411.611} C_VEL
LIN {X 0,Y 320.013,Z 1207.768,A -85,B 0,C 180,E1 13408.21,E2 13408.21} C_VEL
LIN {X 0,Y 320.178,Z 1206.425,A -85,B 0,C 180,E1 13404.265,E2 13404.265} C_VEL
LIN {X 0,Y 320.728,Z 1203.738,A -85,B 0,C 180,E1 13400.49,E2 13400.49} C_VEL
LIN {X 0,Y 322.078,Z 1199.177,A -85,B 0,C 180,E1 13396.34,E2 13396.34} C_VEL
LIN {X 0,Y 324.342,Z 1193.25,A -85,B 0,C 180,E1 13392.416,E2 13392.416} C_VEL
LIN {X 0,Y 327.718,Z 1185.451,A -85,B 0,C 180,E1 13388.524,E2 13388.524} C_VEL
LIN {X 0,Y 332.312,Z 1175.833,A -85,B 0,C 180,E1 13384.707,E2 13384.707} C_VEL
LIN {X 0,Y 337.581,Z 1165.272,A -85,B 0,C 180,E1 13381.327,E2 13381.327} C_VEL
LIN {X 0,Y 343.606,Z 1153.229,A -85,B 0,C 180,E1 13378.182,E2 13378.182} C_VEL
LIN {X 0,Y 350.124,Z 1140.172,A -85,B 0,C 180,E1 13375.334,E2 13375.334} C_VEL
LIN {X 0,Y 356.92,Z 1125.834,A -85,B 0,C 180,E1 13372.765,E2 13372.765} C_VEL
LIN {X 0,Y 364.5,Z 1109.153,A -85,B 0,C 180,E1 13370.272,E2 13370.272} C_VEL
LIN {X 0,Y 371.232,Z 1093.206,A -85,B 0,C 180,E1 13368.298,E2 13368.298} C_VEL
LIN {X 0,Y 378.534,Z 1074.37,A -85,B 0,C 180,E1 13366.367,E2 13366.367} C_VEL
LIN {X 0,Y 385.164,Z 1055.481,A -85,B 0,C 180,E1 13364.766,E2 13364.766} C_VEL
LIN {X 0,Y 391.079,Z 1036.108,A -85,B 0,C 180,E1 13363.44,E2 13363.44} C_VEL
LIN {X 0,Y 396.635,Z 1015.315,A -85,B 0,C 180,E1 13362.28,E2 13362.28} C_VEL
LIN {X 0,Y 401.157,Z 994.882,A -85,B 0,C 180,E1 13361.39,E2 13361.39} C_VEL
LIN {X 0,Y 405.322,Z 971.296,A -85,B 0,C 180,E1 13360.616,E2 13360.616} C_VEL
LIN {X 0,Y 405.743,Z 968.452,A -85,B 0,C 180,E1 13360.54,E2 13360.54} C_VEL
LIN {X 0,Y 406.255,Z 962.04,A -85,B 0,C 180,E1 13360.295,E2 13360.295} C_VEL
LIN {X 0,Y 404.427,Z 941.355,A -85,B 0,C 180,E1 13359.122,E2 13359.122} C_VEL
LIN {X 0,Y 404.467,Z 934.851,A -85,B 0,C 180,E1 13358.916,E2 13358.916} C_VEL
LIN {X 0,Y 417.05,Z 727.873,A -85,B 0,C 180,E1 13355.552,E2 13355.552} C_VEL
LIN {X 0,Y 414.143,Z 689.143,A -85,B 0,C 180,E1 13353.69,E2 13353.69} C_VEL
LIN {X 0,Y 405.81,Z 673.069,A -85,B 0,C 180,E1 13351.036,E2 13351.036} C_VEL
LIN {X 0,Y 399.214,Z 661.253,A -85,B 0,C 180,E1 13348.703,E2 13348.703} C_VEL
LIN {X 0,Y 392.01,Z 648.82,A -85,B 0,C 180,E1 13345.808,E2 13345.808} C_VEL
LIN {X 0,Y 385.696,Z 638.729,A -85,B 0,C 180,E1 13342.884,E2 13342.884} C_VEL
LIN {X 0,Y 380.807,Z 630.947,A -85,B 0,C 180,E1 13340.199,E2 13340.199} C_VEL
LIN {X 0,Y 375.64,Z 622.874,A -85,B 0,C 180,E1 13336.707,E2 13336.707} C_VEL
LIN {X 0,Y 373.038,Z 618.87,A -85,B 0,C 180,E1 13334.514,E2 13334.514} C_VEL
LIN {X 0,Y 370.433,Z 614.641,A -85,B 0,C 180,E1 13331.68,E2 13331.68} C_VEL
LIN {X 0,Y 368.136,Z 610.298,A -85,B 0,C 180,E1 13327.648,E2 13327.648} C_VEL
LIN {X 0,Y 367.43,Z 608.377,A -85,B 0,C 180,E1 13322.183,E2 13322.183} C_VEL
LIN {X 0,Y 368.696,Z 608.724,A -85,B 0,C 180,E1 13318.446,E2 13318.446} C_VEL
LIN {X 0,Y 373.477,Z 612.368,A -85,B 0,C 180,E1 13312.617,E2 13312.617} C_VEL
LIN {X 0,Y 377.649,Z 617.123,A -85,B 0,C 180,E1 13309.319,E2 13309.319} C_VEL
LIN {X 0,Y 379.317,Z 619.043,A -85,B 0,C 180,E1 13308.212,E2 13308.212} C_VEL
LIN {X 0,Y 383.813,Z 624.168,A -85,B 0,C 180,E1 13305.594,E2 13305.594} C_VEL
LIN {X 0,Y 388.929,Z 630.483,A -85,B 0,C 180,E1 13303.034,E2 13303.034} C_VEL
LIN {X 0,Y 394.872,Z 637.952,A -85,B 0,C 180,E1 13300.473,E2 13300.473} C_VEL
LIN {X 0,Y 402.41,Z 648.331,A -85,B 0,C 180,E1 13297.617,E2 13297.617} C_VEL
LIN {X 0,Y 409.892,Z 659.231,A -85,B 0,C 180,E1 13295.115,E2 13295.115} C_VEL
LIN {X 0,Y 418.222,Z 672.419,A -85,B 0,C 180,E1 13292.598,E2 13292.598} C_VEL
LIN {X 0,Y 422.304,Z 679.466,A -85,B 0,C 180,E1 13291.444,E2 13291.444} C_VEL
LIN {X 0,Y 405.1,Z 920.319,A -85,B 0,C 180,E1 13287.229,E2 13287.229} C_VEL
LIN {X 0,Y 402.806,Z 942.672,A -85,B 0,C 180,E1 13286.739,E2 13286.739} C_VEL
LIN {X 0,Y 399.062,Z 967.807,A -85,B 0,C 180,E1 13285.981,E2 13285.981} C_VEL
LIN {X 0,Y 395.151,Z 988.203,A -85,B 0,C 180,E1 13285.18,E2 13285.18} C_VEL
LIN {X 0,Y 389.792,Z 1011.431,A -85,B 0,C 180,E1 13284.025,E2 13284.025} C_VEL
LIN {X 0,Y 384.26,Z 1031.884,A -85,B 0,C 180,E1 13282.771,E2 13282.771} C_VEL
LIN {X 0,Y 377.257,Z 1054.435,A -85,B 0,C 180,E1 13281.086,E2 13281.086} C_VEL
LIN {X 0,Y 370.496,Z 1074.054,A -85,B 0,C 180,E1 13279.317,E2 13279.317} C_VEL
LIN {X 0,Y 363.095,Z 1093.484,A -85,B 0,C 180,E1 13277.211,E2 13277.211} C_VEL
LIN {X 0,Y 355.716,Z 1111.713,A -85,B 0,C 180,E1 13274.871,E2 13274.871} C_VEL
LIN {X 0,Y 348.18,Z 1129.072,A -85,B 0,C 180,E1 13272.19,E2 13272.19} C_VEL
LIN {X 0,Y 341.083,Z 1145.042,A -85,B 0,C 180,E1 13269.286,E2 13269.286} C_VEL
LIN {X 0,Y 334.395,Z 1159.622,A -85,B 0,C 180,E1 13266.089,E2 13266.089} C_VEL
LIN {X 0,Y 328.379,Z 1173.051,A -85,B 0,C 180,E1 13262.611,E2 13262.611} C_VEL
LIN {X 0,Y 323.359,Z 1184.47,A -85,B 0,C 180,E1 13259.042,E2 13259.042} C_VEL
LIN {X 0,Y 319.022,Z 1195.221,A -85,B 0,C 180,E1 13255.031,E2 13255.031} C_VEL
LIN {X 0,Y 315.97,Z 1203.653,A -85,B 0,C 180,E1 13251.146,E2 13251.146} C_VEL
LIN {X 0,Y 313.746,Z 1211.204,A -85,B 0,C 180,E1 13246.858,E2 13246.858} C_VEL
LIN {X 0,Y 312.58,Z 1216.448,A -85,B 0,C 180,E1 13242.939,E2 13242.939} C_VEL
LIN {X 0,Y 312.074,Z 1220.376,A -85,B 0,C 180,E1 13239.032,E2 13239.032} C_VEL
LIN {X 0,Y 311.945,Z 1222.93,A -85,B 0,C 180,E1 13234.965,E2 13234.965} C_VEL
LIN {X 0,Y 311.976,Z 1223.937,A -85,B 0,C 180,E1 13231.469,E2 13231.469} C_VEL
LIN {X 0,Y 311.973,Z 1223.885,A -85,B 0,C 180,E1 13228.163,E2 13228.163} C_VEL
LIN {X 0,Y 311.959,Z 1222.516,A -85,B 0,C 180,E1 13224.113,E2 13224.113} C_VEL
LIN {X 0,Y 312.129,Z 1219.677,A -85,B 0,C 180,E1 13220.225,E2 13220.225} C_VEL
LIN {X 0,Y 312.705,Z 1215.764,A -85,B 0,C 180,E1 13216.502,E2 13216.502} C_VEL
LIN {X 0,Y 314.22,Z 1209.339,A -85,B 0,C 180,E1 13212.022,E2 13212.022} C_VEL
LIN {X 0,Y 316.474,Z 1202.12,A -85,B 0,C 180,E1 13208.111,E2 13208.111} C_VEL
LIN {X 0,Y 320.092,Z 1192.388,A -85,B 0,C 180,E1 13203.868,E2 13203.868} C_VEL
LIN {X 0,Y 324.275,Z 1182.256,A -85,B 0,C 180,E1 13200.237,E2 13200.237} C_VEL
LIN {X 0,Y 330.059,Z 1169.091,A -85,B 0,C 180,E1 13196.333,E2 13196.333} C_VEL
LIN {X 0,Y 336.058,Z 1155.892,A -85,B 0,C 180,E1 13193.059,E2 13193.059} C_VEL
LIN {X 0,Y 342.966,Z 1140.577,A -85,B 0,C 180,E1 13189.888,E2 13189.888} C_VEL
LIN {X 0,Y 350.066,Z 1124.643,A -85,B 0,C 180,E1 13187.094,E2 13187.094} C_VEL
LIN {X 0,Y 357.53,Z 1106.969,A -85,B 0,C 180,E1 13184.51,E2 13184.51} C_VEL
LIN {X 0,Y 365.072,Z 1088.267,A -85,B 0,C 180,E1 13182.197,E2 13182.197} C_VEL
LIN {X 0,Y 372.316,Z 1068.534,A -85,B 0,C 180,E1 13180.18,E2 13180.18} C_VEL
LIN {X 0,Y 379.41,Z 1047.508,A -85,B 0,C 180,E1 13178.376,E2 13178.376} C_VEL
LIN {X 0,Y 385.386,Z 1027.435,A -85,B 0,C 180,E1 13176.957,E2 13176.957} C_VEL
LIN {X 0,Y 391.291,Z 1004.838,A -85,B 0,C 180,E1 13175.635,E2 13175.635} C_VEL
LIN {X 0,Y 396.053,Z 983.009,A -85,B 0,C 180,E1 13174.613,E2 13174.613} C_VEL
LIN {X 0,Y 400.572,Z 957.467,A -85,B 0,C 180,E1 13173.69,E2 13173.69} C_VEL
LIN {X 0,Y 403.614,Z 934.573,A -85,B 0,C 180,E1 13173.078,E2 13173.078} C_VEL
LIN {X 0,Y 406.494,Z 898.868,A -85,B 0,C 180,E1 13172.399,E2 13172.399} C_VEL
LIN {X 0,Y 422.168,Z 679.158,A -85,B 0,C 180,E1 13168.564,E2 13168.564} C_VEL
LIN {X 0,Y 412.879,Z 663.923,A -85,B 0,C 180,E1 13165.882,E2 13165.882} C_VEL
LIN {X 0,Y 403.825,Z 650.319,A -85,B 0,C 180,E1 13162.953,E2 13162.953} C_VEL
LIN {X 0,Y 395.756,Z 639.274,A -85,B 0,C 180,E1 13159.981,E2 13159.981} C_VEL
LIN {X 0,Y 389.48,Z 631.162,A -85,B 0,C 180,E1 13157.326,E2 13157.326} C_VEL
LIN {X 0,Y 384.921,Z 625.646,A -85,B 0,C 180,E1 13155.133,E2 13155.133} C_VEL
LIN {X 0,Y 381.863,Z 621.929,A -85,B 0,C 180,E1 13153.476,E2 13153.476} C_VEL
LIN {X 0,Y 377.83,Z 617.268,A -85,B 0,C 180,E1 13150.984,E2 13150.984} C_VEL
LIN {X 0,Y 373.016,Z 612.038,A -85,B 0,C 180,E1 13147.238,E2 13147.238} C_VEL
LIN {X 0,Y 368.556,Z 608.476,A -85,B 0,C 180,E1 13141.866,E2 13141.866} C_VEL
LIN {X 0,Y 367.168,Z 607.933,A -85,B 0,C 180,E1 13138.127,E2 13138.127} C_VEL
LIN {X 0,Y 367.472,Z 609.589,A -85,B 0,C 180,E1 13133.124,E2 13133.124} C_VEL
LIN {X 0,Y 368.214,Z 610.845,A -85,B 0,C 180,E1 13131.27,E2 13131.27} C_VEL
LIN {X 0,Y 370.949,Z 615.657,A -85,B 0,C 180,E1 13127.23,E2 13127.23} C_VEL
LIN {X 0,Y 374.222,Z 620.81,A -85,B 0,C 180,E1 13124.105,E2 13124.105} C_VEL
LIN {X 0,Y 376.977,Z 625.201,A -85,B 0,C 180,E1 13122.001,E2 13122.001} C_VEL
LIN {X 0,Y 382.057,Z 632.982,A -85,B 0,C 180,E1 13118.828,E2 13118.828} C_VEL
LIN {X 0,Y 388.316,Z 643.054,A -85,B 0,C 180,E1 13115.629,E2 13115.629} C_VEL
LIN {X 0,Y 394.084,Z 652.643,A -85,B 0,C 180,E1 13113.111,E2 13113.111} C_VEL
LIN {X 0,Y 401.018,Z 664.492,A -85,B 0,C 180,E1 13110.458,E2 13110.458} C_VEL
LIN {X 0,Y 408.743,Z 678.774,A -85,B 0,C 180,E1 13107.832,E2 13107.832} C_VEL
LIN {X 0,Y 414.033,Z 689.317,A -85,B 0,C 180,E1 13106.183,E2 13106.183} C_VEL
LIN {X 0,Y 416.889,Z 729.468,A -85,B 0,C 180,E1 13104.29,E2 13104.29} C_VEL
LIN {X 0,Y 403.425,Z 946.16,A -85,B 0,C 180,E1 13100.771,E2 13100.771} C_VEL
LIN {X 0,Y 400.611,Z 969.173,A -85,B 0,C 180,E1 13100.239,E2 13100.239} C_VEL
LIN {X 0,Y 396.801,Z 991.182,A -85,B 0,C 180,E1 13099.55,E2 13099.55} C_VEL
LIN {X 0,Y 392.176,Z 1011.957,A -85,B 0,C 180,E1 13098.674,E2 13098.674} C_VEL
LIN {X 0,Y 386.142,Z 1034.56,A -85,B 0,C 180,E1 13097.449,E2 13097.449} C_VEL
LIN {X 0,Y 380.061,Z 1054.125,A -85,B 0,C 180,E1 13096.123,E2 13096.123} C_VEL
LIN {X 0,Y 373.383,Z 1072.84,A -85,B 0,C 180,E1 13094.555,E2 13094.555} C_VEL
LIN {X 0,Y 366.265,Z 1090.995,A -85,B 0,C 180,E1 13092.727,E2 13092.727} C_VEL
LIN {X 0,Y 359.007,Z 1107.743,A -85,B 0,C 180,E1 13090.67,E2 13090.67} C_VEL
LIN {X 0,Y 351.141,Z 1124.666,A -85,B 0,C 180,E1 13088.163,E2 13088.163} C_VEL
LIN {X 0,Y 343.827,Z 1139.594,A -85,B 0,C 180,E1 13085.484,E2 13085.484} C_VEL
LIN {X 0,Y 336.826,Z 1153.183,A -85,B 0,C 180,E1 13082.499,E2 13082.499} C_VEL
LIN {X 0,Y 330.308,Z 1165.717,A -85,B 0,C 180,E1 13079.167,E2 13079.167} C_VEL
LIN {X 0,Y 325.097,Z 1175.752,A -85,B 0,C 180,E1 13075.895,E2 13075.895} C_VEL
LIN {X 0,Y 320.229,Z 1185.487,A -85,B 0,C 180,E1 13071.972,E2 13071.972} C_VEL
LIN {X 0,Y 316.682,Z 1193.274,A -85,B 0,C 180,E1 13068.024,E2 13068.024} C_VEL
LIN {X 0,Y 314.237,Z 1199.304,A -85,B 0,C 180,E1 13063.951,E2 13063.951} C_VEL
LIN {X 0,Y 312.764,Z 1203.995,A -85,B 0,C 180,E1 13059.569,E2 13059.569} C_VEL
LIN {X 0,Y 312.186,Z 1206.667,A -85,B 0,C 180,E1 13055.698,E2 13055.698} C_VEL
LIN {X 0,Y 312.015,Z 1207.979,A -85,B 0,C 180,E1 13051.653,E2 13051.653} C_VEL
LIN {X 0,Y 312.016,Z 1207.973,A -85,B 0,C 180,E1 13048.164,E2 13048.164} C_VEL
LIN {X 0,Y 312.194,Z 1206.631,A -85,B 0,C 180,E1 13044.118,E2 13044.118} C_VEL
LIN {X 0,Y 312.789,Z 1203.944,A -85,B 0,C 180,E1 13040.246,E2 13040.246} C_VEL
LIN {X 0,Y 314.301,Z 1199.164,A -85,B 0,C 180,E1 13035.821,E2 13035.821} C_VEL
LIN {X 0,Y 316.759,Z 1193.165,A -85,B 0,C 180,E1 13031.79,E2 13031.79} C_VEL
LIN {X 0,Y 320.371,Z 1185.28,A -85,B 0,C 180,E1 13027.813,E2 13027.813} C_VEL
LIN {X 0,Y 325.429,Z 1175.193,A -85,B 0,C 180,E1 13023.79,E2 13023.79} C_VEL
LIN {X 0,Y 331.092,Z 1164.391,A -85,B 0,C 180,E1 13020.313,E2 13020.313} C_VEL
LIN {X 0,Y 337.394,Z 1152.25,A -85,B 0,C 180,E1 13017.159,E2 13017.159} C_VEL
LIN {X 0,Y 344.621,Z 1138.137,A -85,B 0,C 180,E1 13014.122,E2 13014.122} C_VEL
LIN {X 0,Y 351.864,Z 1123.416,A -85,B 0,C 180,E1 13011.515,E2 13011.515} C_VEL
LIN {X 0,Y 359.547,Z 1106.78,A -85,B 0,C 180,E1 13009.088,E2 13009.088} C_VEL
LIN {X 0,Y 366.958,Z 1089.638,A -85,B 0,C 180,E1 13007.009,E2 13007.009} C_VEL
LIN {X 0,Y 374.094,Z 1071.305,A -85,B 0,C 180,E1 13005.192,E2 13005.192} C_VEL
LIN {X 0,Y 381.272,Z 1050.753,A -85,B 0,C 180,E1 13003.523,E2 13003.523} C_VEL
LIN {X 0,Y 387.418,Z 1030.776,A -85,B 0,C 180,E1 13002.209,E2 13002.209} C_VEL
LIN {X 0,Y 392.846,Z 1009.786,A -85,B 0,C 180,E1 13001.117,E2 13001.117} C_VEL
LIN {X 0,Y 397.6,Z 987.803,A -85,B 0,C 180,E1 13000.223,E2 13000.223} C_VEL
LIN {X 0,Y 401.182,Z 966.462,A -85,B 0,C 180,E1 12999.582,E2 12999.582} C_VEL
LIN {X 0,Y 403.848,Z 942.779,A -85,B 0,C 180,E1 12999.061,E2 12999.061} C_VEL
LIN {X 0,Y 404.467,Z 934.851,A -85,B 0,C 180,E1 12998.916,E2 12998.916} C_VEL
LIN {X 0,Y 404.396,Z 927.282,A -85,B 0,C 180,E1 12998.67,E2 12998.67} C_VEL
LIN {X 0,Y 401.938,Z 907.496,A -85,B 0,C 180,E1 12997.627,E2 12997.627} C_VEL
LIN {X 0,Y 401.889,Z 900.978,A -85,B 0,C 180,E1 12997.432,E2 12997.432} C_VEL
LIN {X 0,Y 412.728,Z 729.353,A -85,B 0,C 180,E1 12994.634,E2 12994.634} C_VEL
LIN {X 0,Y 410.246,Z 693.835,A -85,B 0,C 180,E1 12992.903,E2 12992.903} C_VEL
LIN {X 0,Y 402.115,Z 677.818,A -85,B 0,C 180,E1 12990.193,E2 12990.193} C_VEL
LIN {X 0,Y 395.05,Z 664.98,A -85,B 0,C 180,E1 12987.552,E2 12987.552} C_VEL
LIN {X 0,Y 388.579,Z 653.957,A -85,B 0,C 180,E1 12984.799,E2 12984.799} C_VEL
LIN {X 0,Y 383.744,Z 645.897,A -85,B 0,C 180,E1 12982.441,E2 12982.441} C_VEL
LIN {X 0,Y 379.112,Z 638.333,A -85,B 0,C 180,E1 12979.811,E2 12979.811} C_VEL
LIN {X 0,Y 374.197,Z 630.44,A -85,B 0,C 180,E1 12976.374,E2 12976.374} C_VEL
LIN {X 0,Y 371.749,Z 626.578,A -85,B 0,C 180,E1 12974.247,E2 12974.247} C_VEL
LIN {X 0,Y 369.351,Z 622.529,A -85,B 0,C 180,E1 12971.556,E2 12971.556} C_VEL
LIN {X 0,Y 367.113,Z 618.192,A -85,B 0,C 180,E1 12967.512,E2 12967.512} C_VEL
LIN {X 0,Y 366.455,Z 616.32,A -85,B 0,C 180,E1 12962.189,E2 12962.189} C_VEL
LIN {X 0,Y 367.711,Z 616.671,A -85,B 0,C 180,E1 12958.442,E2 12958.442} C_VEL
LIN {X 0,Y 372.318,Z 620.272,A -85,B 0,C 180,E1 12952.749,E2 12952.749} C_VEL
LIN {X 0,Y 376.44,Z 625,A -85,B 0,C 180,E1 12949.439,E2 12949.439} C_VEL
LIN {X 0,Y 382.141,Z 631.692,A -85,B 0,C 180,E1 12945.916,E2 12945.916} C_VEL
LIN {X 0,Y 387.313,Z 638.193,A -85,B 0,C 180,E1 12943.271,E2 12943.271} C_VEL
LIN {X 0,Y 393.083,Z 645.667,A -85,B 0,C 180,E1 12940.728,E2 12940.728} C_VEL
LIN {X 0,Y 400.346,Z 655.836,A -85,B 0,C 180,E1 12937.921,E2 12937.921} C_VEL
LIN {X 0,Y 407.508,Z 666.554,A -85,B 0,C 180,E1 12935.463,E2 12935.463} C_VEL
LIN {X 0,Y 415.622,Z 679.642,A -85,B 0,C 180,E1 12932.955,E2 12932.955} C_VEL
LIN {X 0,Y 417.811,Z 683.685,A -85,B 0,C 180,E1 12932.306,E2 12932.306} C_VEL
LIN {X 0,Y 400.243,Z 922.939,A -85,B 0,C 180,E1 12928.108,E2 12928.108} C_VEL
LIN {X 0,Y 397.789,Z 945.605,A -85,B 0,C 180,E1 12927.598,E2 12927.598} C_VEL
LIN {X 0,Y 394.081,Z 969.139,A -85,B 0,C 180,E1 12926.87,E2 12926.87} C_VEL
LIN {X 0,Y 389.961,Z 989.96,A -85,B 0,C 180,E1 12926.042,E2 12926.042} C_VEL
LIN {X 0,Y 384.438,Z 1012.927,A -85,B 0,C 180,E1 12924.881,E2 12924.881} C_VEL
LIN {X 0,Y 378.448,Z 1034.365,A -85,B 0,C 180,E1 12923.548,E2 12923.548} C_VEL
LIN {X 0,Y 371.565,Z 1055.608,A -85,B 0,C 180,E1 12921.927,E2 12921.927} C_VEL
LIN {X 0,Y 364.351,Z 1075.881,A -85,B 0,C 180,E1 12920.074,E2 12920.074} C_VEL
LIN {X 0,Y 356.704,Z 1095.129,A -85,B 0,C 180,E1 12917.937,E2 12917.937} C_VEL
LIN {X 0,Y 348.953,Z 1113.506,A -85,B 0,C 180,E1 12915.517,E2 12915.517} C_VEL
LIN {X 0,Y 341.489,Z 1130.051,A -85,B 0,C 180,E1 12912.902,E2 12912.902} C_VEL
LIN {X 0,Y 333.914,Z 1146.345,A -85,B 0,C 180,E1 12909.851,E2 12909.851} C_VEL
LIN {X 0,Y 327.375,Z 1160.075,A -85,B 0,C 180,E1 12906.771,E2 12906.771} C_VEL
LIN {X 0,Y 320.783,Z 1174.09,A -85,B 0,C 180,E1 12903.02,E2 12903.02} C_VEL
LIN {X 0,Y 315.661,Z 1185.294,A -85,B 0,C 180,E1 12899.404,E2 12899.404} C_VEL
LIN {X 0,Y 311.007,Z 1196.262,A -85,B 0,C 180,E1 12895.111,E2 12895.111} C_VEL
LIN {X 0,Y 308.036,Z 1204.179,A -85,B 0,C 180,E1 12891.312,E2 12891.312} C_VEL
LIN {X 0,Y 305.678,Z 1211.792,A -85,B 0,C 180,E1 12886.729,E2 12886.729} C_VEL
LIN {X 0,Y 304.566,Z 1216.671,A -85,B 0,C 180,E1 12882.899,E2 12882.899} C_VEL
LIN {X 0,Y 304.038,Z 1220.757,A -85,B 0,C 180,E1 12878.51,E2 12878.51} C_VEL
LIN {X 0,Y 303.954,Z 1222.91,A -85,B 0,C 180,E1 12874.615,E2 12874.615} C_VEL
LIN {X 0,Y 303.978,Z 1223.781,A -85,B 0,C 180,E1 12871.131,E2 12871.131} C_VEL
LIN {X 0,Y 303.958,Z 1223.582,A -85,B 0,C 180,E1 12867.36,E2 12867.36} C_VEL
LIN {X 0,Y 303.985,Z 1221.827,A -85,B 0,C 180,E1 12863.2,E2 12863.2} C_VEL
LIN {X 0,Y 304.186,Z 1219.129,A -85,B 0,C 180,E1 12859.585,E2 12859.585} C_VEL
LIN {X 0,Y 305.024,Z 1214.512,A -85,B 0,C 180,E1 12855.248,E2 12855.248} C_VEL
LIN {X 0,Y 306.7,Z 1208.163,A -85,B 0,C 180,E1 12850.974,E2 12850.974} C_VEL
LIN {X 0,Y 309.403,Z 1200.413,A -85,B 0,C 180,E1 12846.781,E2 12846.781} C_VEL
LIN {X 0,Y 313.267,Z 1190.717,A -85,B 0,C 180,E1 12842.638,E2 12842.638} C_VEL
LIN {X 0,Y 318.13,Z 1179.8,A -85,B 0,C 180,E1 12838.749,E2 12838.749} C_VEL
LIN {X 0,Y 323.789,Z 1167.511,A -85,B 0,C 180,E1 12835.161,E2 12835.161} C_VEL
LIN {X 0,Y 330.543,Z 1153.354,A -85,B 0,C 180,E1 12831.676,E2 12831.676} C_VEL
LIN {X 0,Y 337.464,Z 1138.531,A -85,B 0,C 180,E1 12828.646,E2 12828.646} C_VEL
LIN {X 0,Y 345.222,Z 1121.634,A -85,B 0,C 180,E1 12825.733,E2 12825.733} C_VEL
LIN {X 0,Y 352.348,Z 1105.277,A -85,B 0,C 180,E1 12823.373,E2 12823.373} C_VEL
LIN {X 0,Y 360.365,Z 1085.782,A -85,B 0,C 180,E1 12821.002,E2 12821.002} C_VEL
LIN {X 0,Y 367.344,Z 1067.297,A -85,B 0,C 180,E1 12819.129,E2 12819.129} C_VEL
LIN {X 0,Y 374.942,Z 1045.083,A -85,B 0,C 180,E1 12817.255,E2 12817.255} C_VEL
LIN {X 0,Y 380.819,Z 1025.727,A -85,B 0,C 180,E1 12815.906,E2 12815.906} C_VEL
LIN {X 0,Y 386.928,Z 1002.454,A -85,B 0,C 180,E1 12814.577,E2 12814.577} C_VEL
LIN {X 0,Y 391.667,Z 981.026,A -85,B 0,C 180,E1 12813.593,E2 12813.593} C_VEL
LIN {X 0,Y 395.947,Z 956.887,A -85,B 0,C 180,E1 12812.739,E2 12812.739} C_VEL
LIN {X 0,Y 399.132,Z 933.247,A -85,B 0,C 180,E1 12812.114,E2 12812.114} C_VEL
LIN {X 0,Y 402.691,Z 887.799,A -85,B 0,C 180,E1 12811.271,E2 12811.271} C_VEL
LIN {X 0,Y 417.652,Z 683.252,A -85,B 0,C 180,E1 12807.694,E2 12807.694} C_VEL
LIN {X 0,Y 408.932,Z 668.846,A -85,B 0,C 180,E1 12805.063,E2 12805.063} C_VEL
LIN {X 0,Y 400.791,Z 656.542,A -85,B 0,C 180,E1 12802.323,E2 12802.323} C_VEL
LIN {X 0,Y 393.446,Z 646.268,A -85,B 0,C 180,E1 12799.523,E2 12799.523} C_VEL
LIN {X 0,Y 387.391,Z 638.32,A -85,B 0,C 180,E1 12796.88,E2 12796.88} C_VEL
LIN {X 0,Y 383.084,Z 633,A -85,B 0,C 180,E1 12794.743,E2 12794.743} C_VEL
LIN {X 0,Y 380.351,Z 629.599,A -85,B 0,C 180,E1 12793.221,E2 12793.221} C_VEL
LIN {X 0,Y 376.392,Z 624.963,A -85,B 0,C 180,E1 12790.717,E2 12790.717} C_VEL
LIN {X 0,Y 371.863,Z 619.908,A -85,B 0,C 180,E1 12787.105,E2 12787.105} C_VEL
LIN {X 0,Y 367.486,Z 616.367,A -85,B 0,C 180,E1 12781.715,E2 12781.715} C_VEL
LIN {X 0,Y 366.193,Z 615.875,A -85,B 0,C 180,E1 12778.122,E2 12778.122} C_VEL
LIN {X 0,Y 366.5,Z 617.561,A -85,B 0,C 180,E1 12773.105,E2 12773.105} C_VEL
LIN {X 0,Y 367.17,Z 618.774,A -85,B 0,C 180,E1 12771.386,E2 12771.386} C_VEL
LIN {X 0,Y 369.779,Z 623.498,A -85,B 0,C 180,E1 12767.428,E2 12767.428} C_VEL
LIN {X 0,Y 372.982,Z 628.67,A -85,B 0,C 180,E1 12764.29,E2 12764.29} C_VEL
LIN {X 0,Y 375.485,Z 632.769,A -85,B 0,C 180,E1 12762.327,E2 12762.327} C_VEL
LIN {X 0,Y 380.383,Z 640.495,A -85,B 0,C 180,E1 12759.174,E2 12759.174} C_VEL
LIN {X 0,Y 386.291,Z 650.219,A -85,B 0,C 180,E1 12756.062,E2 12756.062} C_VEL
LIN {X 0,Y 391.929,Z 659.842,A -85,B 0,C 180,E1 12753.524,E2 12753.524} C_VEL
LIN {X 0,Y 398.65,Z 671.57,A -85,B 0,C 180,E1 12750.883,E2 12750.883} C_VEL
LIN {X 0,Y 406.268,Z 686.075,A -85,B 0,C 180,E1 12748.218,E2 12748.218} C_VEL
LIN {X 0,Y 410.151,Z 694.188,A -85,B 0,C 180,E1 12746.959,E2 12746.959} C_VEL
LIN {X 0,Y 412.552,Z 731.038,A -85,B 0,C 180,E1 12745.205,E2 12745.205} C_VEL
LIN {X 0,Y 398.758,Z 945.885,A -85,B 0,C 180,E1 12741.704,E2 12741.704} C_VEL
LIN {X 0,Y 395.875,Z 968.95,A -85,B 0,C 180,E1 12741.171,E2 12741.171} C_VEL
LIN {X 0,Y 392.018,Z 990.771,A -85,B 0,C 180,E1 12740.492,E2 12740.492} C_VEL
LIN {X 0,Y 387.251,Z 1011.703,A -85,B 0,C 180,E1 12739.612,E2 12739.612} C_VEL
LIN {X 0,Y 381.097,Z 1034.229,A -85,B 0,C 180,E1 12738.394,E2 12738.394} C_VEL
LIN {X 0,Y 374.855,Z 1053.819,A -85,B 0,C 180,E1 12737.069,E2 12737.069} C_VEL
LIN {X 0,Y 367.918,Z 1072.779,A -85,B 0,C 180,E1 12735.479,E2 12735.479} C_VEL
LIN {X 0,Y 360.529,Z 1091.101,A -85,B 0,C 180,E1 12733.626,E2 12733.626} C_VEL
LIN {X 0,Y 353.188,Z 1107.553,A -85,B 0,C 180,E1 12731.595,E2 12731.595} C_VEL
LIN {X 0,Y 344.834,Z 1124.975,A -85,B 0,C 180,E1 12728.991,E2 12728.991} C_VEL
LIN {X 0,Y 337.435,Z 1139.565,A -85,B 0,C 180,E1 12726.343,E2 12726.343} C_VEL
LIN {X 0,Y 330.39,Z 1152.763,A -85,B 0,C 180,E1 12723.421,E2 12723.421} C_VEL
LIN {X 0,Y 323.754,Z 1165.063,A -85,B 0,C 180,E1 12720.144,E2 12720.144} C_VEL
LIN {X 0,Y 318.077,Z 1175.486,A -85,B 0,C 180,E1 12716.712,E2 12716.712} C_VEL
LIN {X 0,Y 312.954,Z 1185.252,A -85,B 0,C 180,E1 12712.742,E2 12712.742} C_VEL
LIN {X 0,Y 309.126,Z 1193.172,A -85,B 0,C 180,E1 12708.676,E2 12708.676} C_VEL
LIN {X 0,Y 306.503,Z 1199.218,A -85,B 0,C 180,E1 12704.548,E2 12704.548} C_VEL
LIN {X 0,Y 304.919,Z 1203.9,A -85,B 0,C 180,E1 12700.199,E2 12700.199} C_VEL
LIN {X 0,Y 304.236,Z 1206.659,A -85,B 0,C 180,E1 12696.226,E2 12696.226} C_VEL
LIN {X 0,Y 304.028,Z 1208.141,A -85,B 0,C 180,E1 12692.073,E2 12692.073} C_VEL
LIN {X 0,Y 304.013,Z 1208.219,A -85,B 0,C 180,E1 12688.492,E2 12688.492} C_VEL
LIN {X 0,Y 304.164,Z 1207.154,A -85,B 0,C 180,E1 12684.53,E2 12684.53} C_VEL
LIN {X 0,Y 304.757,Z 1204.453,A -85,B 0,C 180,E1 12680.368,E2 12680.368} C_VEL
LIN {X 0,Y 306.201,Z 1200.102,A -85,B 0,C 180,E1 12676.017,E2 12676.017} C_VEL
LIN {X 0,Y 308.639,Z 1194.255,A -85,B 0,C 180,E1 12671.881,E2 12671.881} C_VEL
LIN {X 0,Y 312.272,Z 1186.67,A -85,B 0,C 180,E1 12667.801,E2 12667.801} C_VEL
LIN {X 0,Y 316.945,Z 1177.779,A -85,B 0,C 180,E1 12663.992,E2 12663.992} C_VEL
LIN {X 0,Y 322.81,Z 1166.856,A -85,B 0,C 180,E1 12660.292,E2 12660.292} C_VEL
LIN {X 0,Y 329.881,Z 1153.869,A -85,B 0,C 180,E1 12656.729,E2 12656.729} C_VEL
LIN {X 0,Y 337.277,Z 1140.071,A -85,B 0,C 180,E1 12653.637,E2 12653.637} C_VEL
LIN {X 0,Y 344.662,Z 1125.528,A -85,B 0,C 180,E1 12650.986,E2 12650.986} C_VEL
LIN {X 0,Y 352.832,Z 1108.601,A -85,B 0,C 180,E1 12648.431,E2 12648.431} C_VEL
LIN {X 0,Y 360.187,Z 1092.166,A -85,B 0,C 180,E1 12646.384,E2 12646.384} C_VEL
LIN {X 0,Y 367.798,Z 1073.461,A -85,B 0,C 180,E1 12644.471,E2 12644.471} C_VEL
LIN {X 0,Y 374.788,Z 1054.48,A -85,B 0,C 180,E1 12642.868,E2 12642.868} C_VEL
LIN {X 0,Y 381.19,Z 1034.421,A -85,B 0,C 180,E1 12641.508,E2 12641.508} C_VEL
LIN {X 0,Y 387.268,Z 1012.273,A -85,B 0,C 180,E1 12640.306,E2 12640.306} C_VEL
LIN {X 0,Y 392.116,Z 991.054,A -85,B 0,C 180,E1 12639.41,E2 12639.41} C_VEL
LIN {X 0,Y 396.06,Z 968.813,A -85,B 0,C 180,E1 12638.718,E2 12638.718} C_VEL
LIN {X 0,Y 398.937,Z 945.773,A -85,B 0,C 180,E1 12638.187,E2 12638.187} C_VEL
LIN {X 0,Y 401.889,Z 900.978,A -85,B 0,C 180,E1 12637.432,E2 12637.432} C_VEL
LIN {X 0,Y 401.788,Z 893.4,A -85,B 0,C 180,E1 12637.188,E2 12637.188} C_VEL
LIN {X 0,Y 399.576,Z 873.626,A -85,B 0,C 180,E1 12636.122,E2 12636.122} C_VEL
LIN {X 0,Y 399.59,Z 867.109,A -85,B 0,C 180,E1 12635.927,E2 12635.927} C_VEL
LIN {X 0,Y 408.512,Z 730.845,A -85,B 0,C 180,E1 12633.699,E2 12633.699} C_VEL
LIN {X 0,Y 406.384,Z 698.392,A -85,B 0,C 180,E1 12632.083,E2 12632.083} C_VEL
LIN {X 0,Y 398.951,Z 683.58,A -85,B 0,C 180,E1 12629.504,E2 12629.504} C_VEL
LIN {X 0,Y 392.445,Z 671.43,A -85,B 0,C 180,E1 12626.97,E2 12626.97} C_VEL
LIN {X 0,Y 386.376,Z 660.872,A -85,B 0,C 180,E1 12624.297,E2 12624.297} C_VEL
LIN {X 0,Y 381.815,Z 653.064,A -85,B 0,C 180,E1 12621.993,E2 12621.993} C_VEL
LIN {X 0,Y 377.395,Z 645.656,A -85,B 0,C 180,E1 12619.393,E2 12619.393} C_VEL
LIN {X 0,Y 372.668,Z 637.862,A -85,B 0,C 180,E1 12615.963,E2 12615.963} C_VEL
LIN {X 0,Y 370.47,Z 634.286,A -85,B 0,C 180,E1 12613.979,E2 12613.979} C_VEL
LIN {X 0,Y 368.152,Z 630.273,A -85,B 0,C 180,E1 12611.277,E2 12611.277} C_VEL
LIN {X 0,Y 366.025,Z 626.008,A -85,B 0,C 180,E1 12607.219,E2 12607.219} C_VEL
LIN {X 0,Y 365.504,Z 624.248,A -85,B 0,C 180,E1 12602.038,E2 12602.038} C_VEL
LIN {X 0,Y 366.808,Z 624.67,A -85,B 0,C 180,E1 12598.282,E2 12598.282} C_VEL
LIN {X 0,Y 371.234,Z 628.328,A -85,B 0,C 180,E1 12592.805,E2 12592.805} C_VEL
LIN {X 0,Y 376.086,Z 633.93,A -85,B 0,C 180,E1 12588.964,E2 12588.964} C_VEL
LIN {X 0,Y 380.608,Z 639.396,A -85,B 0,C 180,E1 12586.169,E2 12586.169} C_VEL
LIN {X 0,Y 385.703,Z 645.899,A -85,B 0,C 180,E1 12583.509,E2 12583.509} C_VEL
LIN {X 0,Y 392.044,Z 654.408,A -85,B 0,C 180,E1 12580.675,E2 12580.675} C_VEL
LIN {X 0,Y 399.292,Z 664.763,A -85,B 0,C 180,E1 12577.86,E2 12577.86} C_VEL
LIN {X 0,Y 407.714,Z 677.948,A -85,B 0,C 180,E1 12574.973,E2 12574.973} C_VEL
LIN {X 0,Y 413.43,Z 687.819,A -85,B 0,C 180,E1 12573.187,E2 12573.187} C_VEL
LIN {X 0,Y 395.531,Z 925.035,A -85,B 0,C 180,E1 12569.02,E2 12569.02} C_VEL
LIN {X 0,Y 392.794,Z 948.888,A -85,B 0,C 180,E1 12568.467,E2 12568.467} C_VEL
LIN {X 0,Y 389.056,Z 971.238,A -85,B 0,C 180,E1 12567.753,E2 12567.753} C_VEL
LIN {X 0,Y 384.52,Z 993.328,A -85,B 0,C 180,E1 12566.855,E2 12566.855} C_VEL
LIN {X 0,Y 379.168,Z 1014.443,A -85,B 0,C 180,E1 12565.76,E2 12565.76} C_VEL
LIN {X 0,Y 372.764,Z 1036.563,A -85,B 0,C 180,E1 12564.363,E2 12564.363} C_VEL
LIN {X 0,Y 365.946,Z 1056.808,A -85,B 0,C 180,E1 12562.792,E2 12562.792} C_VEL
LIN {X 0,Y 358.314,Z 1077.432,A -85,B 0,C 180,E1 12560.872,E2 12560.872} C_VEL
LIN {X 0,Y 350.778,Z 1095.796,A -85,B 0,C 180,E1 12558.808,E2 12558.808} C_VEL
LIN {X 0,Y 342.473,Z 1114.726,A -85,B 0,C 180,E1 12556.268,E2 12556.268} C_VEL
LIN {X 0,Y 335.015,Z 1130.681,A -85,B 0,C 180,E1 12553.702,E2 12553.702} C_VEL
LIN {X 0,Y 326.779,Z 1147.647,A -85,B 0,C 180,E1 12550.441,E2 12550.441} C_VEL
LIN {X 0,Y 320.054,Z 1161.247,A -85,B 0,C 180,E1 12547.305,E2 12547.305} C_VEL
LIN {X 0,Y 313.306,Z 1174.928,A -85,B 0,C 180,E1 12543.511,E2 12543.511} C_VEL
LIN {X 0,Y 307.976,Z 1186.121,A -85,B 0,C 180,E1 12539.783,E2 12539.783} C_VEL
LIN {X 0,Y 303.35,Z 1196.454,A -85,B 0,C 180,E1 12535.581,E2 12535.581} C_VEL
LIN {X 0,Y 300.241,Z 1204.313,A -85,B 0,C 180,E1 12531.694,E2 12531.694} C_VEL
LIN {X 0,Y 297.76,Z 1211.845,A -85,B 0,C 180,E1 12526.986,E2 12526.986} C_VEL
LIN {X 0,Y 296.584,Z 1216.725,A -85,B 0,C 180,E1 12523.011,E2 12523.011} C_VEL
LIN {X 0,Y 296.04,Z 1220.671,A -85,B 0,C 180,E1 12518.546,E2 12518.546} C_VEL
LIN {X 0,Y 295.954,Z 1222.729,A -85,B 0,C 180,E1 12514.675,E2 12514.675} C_VEL
LIN {X 0,Y 295.981,Z 1223.576,A -85,B 0,C 180,E1 12511.161,E2 12511.161} C_VEL
LIN {X 0,Y 295.962,Z 1223.402,A -85,B 0,C 180,E1 12507.483,E2 12507.483} C_VEL
LIN {X 0,Y 295.985,Z 1221.74,A -85,B 0,C 180,E1 12503.21,E2 12503.21} C_VEL
LIN {X 0,Y 296.193,Z 1219.088,A -85,B 0,C 180,E1 12499.497,E2 12499.497} C_VEL
LIN {X 0,Y 296.977,Z 1214.902,A -85,B 0,C 180,E1 12495.374,E2 12495.374} C_VEL
LIN {X 0,Y 298.734,Z 1208.578,A -85,B 0,C 180,E1 12490.852,E2 12490.852} C_VEL
LIN {X 0,Y 301.36,Z 1201.301,A -85,B 0,C 180,E1 12486.745,E2 12486.745} C_VEL
LIN {X 0,Y 305.503,Z 1191.433,A -85,B 0,C 180,E1 12482.307,E2 12482.307} C_VEL
LIN {X 0,Y 310.237,Z 1181.231,A -85,B 0,C 180,E1 12478.526,E2 12478.526} C_VEL
LIN {X 0,Y 316.461,Z 1168.348,A -85,B 0,C 180,E1 12474.605,E2 12474.605} C_VEL
LIN {X 0,Y 323.317,Z 1154.621,A -85,B 0,C 180,E1 12471.114,E2 12471.114} C_VEL
LIN {X 0,Y 330.856,Z 1139.093,A -85,B 0,C 180,E1 12467.864,E2 12467.864} C_VEL
LIN {X 0,Y 338.874,Z 1122.325,A -85,B 0,C 180,E1 12464.917,E2 12464.917} C_VEL
LIN {X 0,Y 346.34,Z 1105.771,A -85,B 0,C 180,E1 12462.498,E2 12462.498} C_VEL
LIN {X 0,Y 354.474,Z 1086.701,A -85,B 0,C 180,E1 12460.146,E2 12460.146} C_VEL
LIN {X 0,Y 361.641,Z 1068.307,A -85,B 0,C 180,E1 12458.261,E2 12458.261} C_VEL
LIN {X 0,Y 369.159,Z 1047.175,A -85,B 0,C 180,E1 12456.446,E2 12456.446} C_VEL
LIN {X 0,Y 375.383,Z 1027.331,A -85,B 0,C 180,E1 12455.044,E2 12455.044} C_VEL
LIN {X 0,Y 381.638,Z 1004.474,A -85,B 0,C 180,E1 12453.714,E2 12453.714} C_VEL
LIN {X 0,Y 386.418,Z 983.591,A -85,B 0,C 180,E1 12452.739,E2 12452.739} C_VEL
LIN {X 0,Y 391.165,Z 958.043,A -85,B 0,C 180,E1 12451.816,E2 12451.816} C_VEL
LIN {X 0,Y 394.329,Z 935.302,A -85,B 0,C 180,E1 12451.209,E2 12451.209} C_VEL
LIN {X 0,Y 397.334,Z 900.017,A -85,B 0,C 180,E1 12450.536,E2 12450.536} C_VEL
LIN {X 0,Y 413.275,Z 687.536,A -85,B 0,C 180,E1 12446.822,E2 12446.822} C_VEL
LIN {X 0,Y 405.452,Z 674.475,A -85,B 0,C 180,E1 12444.359,E2 12444.359} C_VEL
LIN {X 0,Y 398.172,Z 663.268,A -85,B 0,C 180,E1 12441.818,E2 12441.818} C_VEL
LIN {X 0,Y 391,Z 653.023,A -85,B 0,C 180,E1 12438.991,E2 12438.991} C_VEL
LIN {X 0,Y 385.473,Z 645.66,A -85,B 0,C 180,E1 12436.501,E2 12436.501} C_VEL
LIN {X 0,Y 379.483,Z 637.902,A -85,B 0,C 180,E1 12433.33,E2 12433.33} C_VEL
LIN {X 0,Y 374.964,Z 632.657,A -85,B 0,C 180,E1 12430.447,E2 12430.447} C_VEL
LIN {X 0,Y 370.547,Z 627.663,A -85,B 0,C 180,E1 12426.819,E2 12426.819} C_VEL
LIN {X 0,Y 366.506,Z 624.317,A -85,B 0,C 180,E1 12421.72,E2 12421.72} C_VEL
LIN {X 0,Y 365.218,Z 623.817,A -85,B 0,C 180,E1 12418.117,E2 12418.117} C_VEL
LIN {X 0,Y 365.528,Z 625.532,A -85,B 0,C 180,E1 12413.087,E2 12413.087} C_VEL
LIN {X 0,Y 366.123,Z 626.682,A -85,B 0,C 180,E1 12411.519,E2 12411.519} C_VEL
LIN {X 0,Y 368.613,Z 631.337,A -85,B 0,C 180,E1 12407.626,E2 12407.626} C_VEL
LIN {X 0,Y 371.658,Z 636.38,A -85,B 0,C 180,E1 12404.553,E2 12404.553} C_VEL
LIN {X 0,Y 374.204,Z 640.694,A -85,B 0,C 180,E1 12402.506,E2 12402.506} C_VEL
LIN {X 0,Y 378.664,Z 647.889,A -85,B 0,C 180,E1 12399.56,E2 12399.56} C_VEL
LIN {X 0,Y 384.36,Z 657.508,A -85,B 0,C 180,E1 12396.464,E2 12396.464} C_VEL
LIN {X 0,Y 389.722,Z 666.893,A -85,B 0,C 180,E1 12393.977,E2 12393.977} C_VEL
LIN {X 0,Y 396.032,Z 678.17,A -85,B 0,C 180,E1 12391.416,E2 12391.416} C_VEL
LIN {X 0,Y 403.38,Z 692.503,A -85,B 0,C 180,E1 12388.756,E2 12388.756} C_VEL
LIN {X 0,Y 406.333,Z 698.889,A -85,B 0,C 180,E1 12387.756,E2 12387.756} C_VEL
LIN {X 0,Y 408.334,Z 732.495,A -85,B 0,C 180,E1 12386.142,E2 12386.142} C_VEL
LIN {X 0,Y 394.201,Z 945.61,A -85,B 0,C 180,E1 12382.66,E2 12382.66} C_VEL
LIN {X 0,Y 391.265,Z 968.593,A -85,B 0,C 180,E1 12382.129,E2 12382.129} C_VEL
LIN {X 0,Y 387.344,Z 990.359,A -85,B 0,C 180,E1 12381.457,E2 12381.457} C_VEL
LIN {X 0,Y 382.466,Z 1011.317,A -85,B 0,C 180,E1 12380.579,E2 12380.579} C_VEL
LIN {X 0,Y 376.472,Z 1032.901,A -85,B 0,C 180,E1 12379.427,E2 12379.427} C_VEL
LIN {X 0,Y 370.055,Z 1052.622,A -85,B 0,C 180,E1 12378.106,E2 12378.106} C_VEL
LIN {X 0,Y 362.711,Z 1072.319,A -85,B 0,C 180,E1 12376.468,E2 12376.468} C_VEL
LIN {X 0,Y 355.153,Z 1090.622,A -85,B 0,C 180,E1 12374.621,E2 12374.621} C_VEL
LIN {X 0,Y 347.465,Z 1107.359,A -85,B 0,C 180,E1 12372.55,E2 12372.55} C_VEL
LIN {X 0,Y 339.077,Z 1124.372,A -85,B 0,C 180,E1 12370.003,E2 12370.003} C_VEL
LIN {X 0,Y 331.384,Z 1139.027,A -85,B 0,C 180,E1 12367.334,E2 12367.334} C_VEL
LIN {X 0,Y 324.043,Z 1152.342,A -85,B 0,C 180,E1 12364.379,E2 12364.379} C_VEL
LIN {X 0,Y 317.23,Z 1164.517,A -85,B 0,C 180,E1 12361.125,E2 12361.125} C_VEL
LIN {X 0,Y 310.906,Z 1175.618,A -85,B 0,C 180,E1 12357.422,E2 12357.422} C_VEL
LIN {X 0,Y 305.485,Z 1185.472,A -85,B 0,C 180,E1 12353.33,E2 12353.33} C_VEL
LIN {X 0,Y 301.454,Z 1193.391,A -85,B 0,C 180,E1 12349.169,E2 12349.169} C_VEL
LIN {X 0,Y 298.678,Z 1199.428,A -85,B 0,C 180,E1 12344.938,E2 12344.938} C_VEL
LIN {X 0,Y 296.99,Z 1204.107,A -85,B 0,C 180,E1 12340.475,E2 12340.475} C_VEL
LIN {X 0,Y 296.256,Z 1206.865,A -85,B 0,C 180,E1 12336.395,E2 12336.395} C_VEL
LIN {X 0,Y 296.031,Z 1208.346,A -85,B 0,C 180,E1 12332.129,E2 12332.129} C_VEL
LIN {X 0,Y 296.016,Z 1208.423,A -85,B 0,C 180,E1 12328.452,E2 12328.452} C_VEL
LIN {X 0,Y 296.179,Z 1207.359,A -85,B 0,C 180,E1 12324.382,E2 12324.382} C_VEL
LIN {X 0,Y 296.822,Z 1204.66,A -85,B 0,C 180,E1 12320.108,E2 12320.108} C_VEL
LIN {X 0,Y 298.357,Z 1200.312,A -85,B 0,C 180,E1 12315.641,E2 12315.641} C_VEL
LIN {X 0,Y 300.943,Z 1194.467,A -85,B 0,C 180,E1 12311.401,E2 12311.401} C_VEL
LIN {X 0,Y 304.811,Z 1186.816,A -85,B 0,C 180,E1 12307.189,E2 12307.189} C_VEL
LIN {X 0,Y 309.669,Z 1178.005,A -85,B 0,C 180,E1 12303.333,E2 12303.333} C_VEL
LIN {X 0,Y 315.466,Z 1167.648,A -85,B 0,C 180,E1 12299.739,E2 12299.739} C_VEL
LIN {X 0,Y 322.386,Z 1155.488,A -85,B 0,C 180,E1 12296.279,E2 12296.279} C_VEL
LIN {X 0,Y 329.524,Z 1142.617,A -85,B 0,C 180,E1 12293.291,E2 12293.291} C_VEL
LIN {X 0,Y 337.492,Z 1127.64,A -85,B 0,C 180,E1 12290.434,E2 12290.434} C_VEL
LIN {X 0,Y 345.512,Z 1111.809,A -85,B 0,C 180,E1 12287.939,E2 12287.939} C_VEL
LIN {X 0,Y 353.33,Z 1094.934,A -85,B 0,C 180,E1 12285.769,E2 12285.769} C_VEL
LIN {X 0,Y 361.096,Z 1076.815,A -85,B 0,C 180,E1 12283.837,E2 12283.837} C_VEL
LIN {X 0,Y 368.184,Z 1058.29,A -85,B 0,C 180,E1 12282.221,E2 12282.221} C_VEL
LIN {X 0,Y 375.036,Z 1038.04,A -85,B 0,C 180,E1 12280.783,E2 12280.783} C_VEL
LIN {X 0,Y 380.951,Z 1017.898,A -85,B 0,C 180,E1 12279.629,E2 12279.629} C_VEL
LIN {X 0,Y 386.138,Z 996.549,A -85,B 0,C 180,E1 12278.676,E2 12278.676} C_VEL
LIN {X 0,Y 390.513,Z 974.495,A -85,B 0,C 180,E1 12277.923,E2 12277.923} C_VEL
LIN {X 0,Y 393.66,Z 952.302,A -85,B 0,C 180,E1 12277.373,E2 12277.373} C_VEL
LIN {X 0,Y 396.085,Z 922.016,A -85,B 0,C 180,E1 12276.823,E2 12276.823} C_VEL
LIN {X 0,Y 399.59,Z 867.109,A -85,B 0,C 180,E1 12275.927,E2 12275.927} C_VEL
LIN {X 0,Y 399.547,Z 859.531,A -85,B 0,C 180,E1 12275.683,E2 12275.683} C_VEL
LIN {X 0,Y 397.514,Z 839.774,A -85,B 0,C 180,E1 12274.594,E2 12274.594} C_VEL
LIN {X 0,Y 397.565,Z 833.257,A -85,B 0,C 180,E1 12274.398,E2 12274.398} C_VEL
LIN {X 0,Y 404.418,Z 732.286,A -85,B 0,C 180,E1 12272.741,E2 12272.741} C_VEL
LIN {X 0,Y 402.652,Z 703.037,A -85,B 0,C 180,E1 12271.266,E2 12271.266} C_VEL
LIN {X 0,Y 394.961,Z 687.593,A -85,B 0,C 180,E1 12268.462,E2 12268.462} C_VEL
LIN {X 0,Y 388.409,Z 675.316,A -85,B 0,C 180,E1 12265.748,E2 12265.748} C_VEL
LIN {X 0,Y 383.839,Z 667.148,A -85,B 0,C 180,E1 12263.61,E2 12263.61} C_VEL
LIN {X 0,Y 379.713,Z 659.897,A -85,B 0,C 180,E1 12261.43,E2 12261.43} C_VEL
LIN {X 0,Y 375.663,Z 652.921,A -85,B 0,C 180,E1 12258.949,E2 12258.949} C_VEL
LIN {X 0,Y 371.157,Z 645.281,A -85,B 0,C 180,E1 12255.548,E2 12255.548} C_VEL
LIN {X 0,Y 369.124,Z 641.887,A -85,B 0,C 180,E1 12253.631,E2 12253.631} C_VEL
LIN {X 0,Y 366.961,Z 638.015,A -85,B 0,C 180,E1 12250.996,E2 12250.996} C_VEL
LIN {X 0,Y 364.997,Z 633.899,A -85,B 0,C 180,E1 12247.081,E2 12247.081} C_VEL
LIN {X 0,Y 364.556,Z 632.177,A -85,B 0,C 180,E1 12241.886,E2 12241.886} C_VEL
LIN {X 0,Y 365.994,Z 632.73,A -85,B 0,C 180,E1 12237.965,E2 12237.965} C_VEL
LIN {X 0,Y 370.075,Z 636.257,A -85,B 0,C 180,E1 12232.938,E2 12232.938} C_VEL
LIN {X 0,Y 374.65,Z 641.611,A -85,B 0,C 180,E1 12229.233,E2 12229.233} C_VEL
LIN {X 0,Y 378.958,Z 646.918,A -85,B 0,C 180,E1 12226.496,E2 12226.496} C_VEL
LIN {X 0,Y 384.84,Z 654.492,A -85,B 0,C 180,E1 12223.393,E2 12223.393} C_VEL
LIN {X 0,Y 391.583,Z 663.943,A -85,B 0,C 180,E1 12220.38,E2 12220.38} C_VEL
LIN {X 0,Y 399.226,Z 675.435,A -85,B 0,C 180,E1 12217.429,E2 12217.429} C_VEL
LIN {X 0,Y 406.5,Z 687.359,A -85,B 0,C 180,E1 12214.932,E2 12214.932} C_VEL
LIN {X 0,Y 409.126,Z 692.099,A -85,B 0,C 180,E1 12214.084,E2 12214.084} C_VEL
LIN {X 0,Y 391.01,Z 926.205,A -85,B 0,C 180,E1 12209.972,E2 12209.972} C_VEL
LIN {X 0,Y 388.107,Z 950.304,A -85,B 0,C 180,E1 12209.405,E2 12209.405} C_VEL
LIN {X 0,Y 384.401,Z 971.875,A -85,B 0,C 180,E1 12208.712,E2 12208.712} C_VEL
LIN {X 0,Y 379.788,Z 993.734,A -85,B 0,C 180,E1 12207.822,E2 12207.822} C_VEL
LIN {X 0,Y 374.1,Z 1015.569,A -85,B 0,C 180,E1 12206.686,E2 12206.686} C_VEL
LIN {X 0,Y 367.428,Z 1037.802,A -85,B 0,C 180,E1 12205.267,E2 12205.267} C_VEL
LIN {X 0,Y 360.443,Z 1057.929,A -85,B 0,C 180,E1 12203.691,E2 12203.691} C_VEL
LIN {X 0,Y 352.188,Z 1079.357,A -85,B 0,C 180,E1 12201.658,E2 12201.658} C_VEL
LIN {X 0,Y 344.593,Z 1097.261,A -85,B 0,C 180,E1 12199.611,E2 12199.611} C_VEL
LIN {X 0,Y 335.804,Z 1116.465,A -85,B 0,C 180,E1 12196.968,E2 12196.968} C_VEL
LIN {X 0,Y 327.929,Z 1132.738,A -85,B 0,C 180,E1 12194.284,E2 12194.284} C_VEL
LIN {X 0,Y 319.787,Z 1148.747,A -85,B 0,C 180,E1 12191.101,E2 12191.101} C_VEL
LIN {X 0,Y 312.409,Z 1163.14,A -85,B 0,C 180,E1 12187.683,E2 12187.683} C_VEL
LIN {X 0,Y 305.801,Z 1175.866,A -85,B 0,C 180,E1 12183.994,E2 12183.994} C_VEL
LIN {X 0,Y 299.993,Z 1187.588,A -85,B 0,C 180,E1 12179.935,E2 12179.935} C_VEL
LIN {X 0,Y 295.34,Z 1197.494,A -85,B 0,C 180,E1 12175.679,E2 12175.679} C_VEL
LIN {X 0,Y 291.925,Z 1205.867,A -85,B 0,C 180,E1 12171.288,E2 12171.288} C_VEL
LIN {X 0,Y 289.689,Z 1212.432,A -85,B 0,C 180,E1 12166.853,E2 12166.853} C_VEL
LIN {X 0,Y 288.462,Z 1217.545,A -85,B 0,C 180,E1 12162.41,E2 12162.41} C_VEL
LIN {X 0,Y 288.008,Z 1220.827,A -85,B 0,C 180,E1 12158.183,E2 12158.183} C_VEL
LIN {X 0,Y 287.957,Z 1222.605,A -85,B 0,C 180,E1 12154.581,E2 12154.581} C_VEL
LIN {X 0,Y 287.978,Z 1223.42,A -85,B 0,C 180,E1 12150.796,E2 12150.796} C_VEL
LIN {X 0,Y 287.961,Z 1223.027,A -85,B 0,C 180,E1 12146.616,E2 12146.616} C_VEL
LIN {X 0,Y 287.982,Z 1221.291,A -85,B 0,C 180,E1 12142.619,E2 12142.619} C_VEL
LIN {X 0,Y 288.273,Z 1218.539,A -85,B 0,C 180,E1 12138.8,E2 12138.8} C_VEL
LIN {X 0,Y 289.327,Z 1213.726,A -85,B 0,C 180,E1 12134.157,E2 12134.157} C_VEL
LIN {X 0,Y 291.199,Z 1207.722,A -85,B 0,C 180,E1 12129.918,E2 12129.918} C_VEL
LIN {X 0,Y 294.293,Z 1199.954,A -85,B 0,C 180,E1 12125.513,E2 12125.513} C_VEL
LIN {X 0,Y 298.412,Z 1190.718,A -85,B 0,C 180,E1 12121.371,E2 12121.371} C_VEL
LIN {X 0,Y 303.744,Z 1179.915,A -85,B 0,C 180,E1 12117.327,E2 12117.327} C_VEL
LIN {X 0,Y 309.954,Z 1167.641,A -85,B 0,C 180,E1 12113.591,E2 12113.591} C_VEL
LIN {X 0,Y 317.275,Z 1153.564,A -85,B 0,C 180,E1 12109.993,E2 12109.993} C_VEL
LIN {X 0,Y 324.855,Z 1138.585,A -85,B 0,C 180,E1 12106.843,E2 12106.843} C_VEL
LIN {X 0,Y 333.107,Z 1121.919,A -85,B 0,C 180,E1 12103.9,E2 12103.9} C_VEL
LIN {X 0,Y 340.869,Z 1105.278,A -85,B 0,C 180,E1 12101.458,E2 12101.458} C_VEL
LIN {X 0,Y 349.497,Z 1085.575,A -85,B 0,C 180,E1 12099.039,E2 12099.039} C_VEL
LIN {X 0,Y 356.611,Z 1067.821,A -85,B 0,C 180,E1 12097.225,E2 12097.225} C_VEL
LIN {X 0,Y 364.54,Z 1045.974,A -85,B 0,C 180,E1 12095.363,E2 12095.363} C_VEL
LIN {X 0,Y 370.82,Z 1026.395,A -85,B 0,C 180,E1 12093.991,E2 12093.991} C_VEL
LIN {X 0,Y 377.274,Z 1003.111,A -85,B 0,C 180,E1 12092.658,E2 12092.658} C_VEL
LIN {X 0,Y 382.014,Z 982.761,A -85,B 0,C 180,E1 12091.72,E2 12091.72} C_VEL
LIN {X 0,Y 386.698,Z 957.884,A -85,B 0,C 180,E1 12090.832,E2 12090.832} C_VEL
LIN {X 0,Y 389.976,Z 934.702,A -85,B 0,C 180,E1 12090.219,E2 12090.219} C_VEL
LIN {X 0,Y 393.281,Z 895.789,A -85,B 0,C 180,E1 12089.486,E2 12089.486} C_VEL
LIN {X 0,Y 408.956,Z 691.67,A -85,B 0,C 180,E1 12085.915,E2 12085.915} C_VEL
LIN {X 0,Y 401.09,Z 678.5,A -85,B 0,C 180,E1 12083.313,E2 12083.313} C_VEL
LIN {X 0,Y 393.493,Z 666.821,A -85,B 0,C 180,E1 12080.489,E2 12080.489} C_VEL
LIN {X 0,Y 386.861,Z 657.439,A -85,B 0,C 180,E1 12077.68,E2 12077.68} C_VEL
LIN {X 0,Y 381.337,Z 649.958,A -85,B 0,C 180,E1 12074.968,E2 12074.968} C_VEL
LIN {X 0,Y 377.104,Z 644.683,A -85,B 0,C 180,E1 12072.558,E2 12072.558} C_VEL
LIN {X 0,Y 373.544,Z 640.349,A -85,B 0,C 180,E1 12070.176,E2 12070.176} C_VEL
LIN {X 0,Y 369.4,Z 635.533,A -85,B 0,C 180,E1 12066.684,E2 12066.684} C_VEL
LIN {X 0,Y 365.449,Z 632.21,A -85,B 0,C 180,E1 12061.568,E2 12061.568} C_VEL
LIN {X 0,Y 364.216,Z 631.773,A -85,B 0,C 180,E1 12057.955,E2 12057.955} C_VEL
LIN {X 0,Y 364.724,Z 633.737,A -85,B 0,C 180,E1 12052.597,E2 12052.597} C_VEL
LIN {X 0,Y 367.275,Z 638.771,A -85,B 0,C 180,E1 12048.059,E2 12048.059} C_VEL
LIN {X 0,Y 370.343,Z 644.089,A -85,B 0,C 180,E1 12044.818,E2 12044.818} C_VEL
LIN {X 0,Y 372.923,Z 648.609,A -85,B 0,C 180,E1 12042.685,E2 12042.685} C_VEL
LIN {X 0,Y 377.139,Z 655.622,A -85,B 0,C 180,E1 12039.839,E2 12039.839} C_VEL
LIN {X 0,Y 382.382,Z 664.673,A -85,B 0,C 180,E1 12036.906,E2 12036.906} C_VEL
LIN {X 0,Y 387.539,Z 673.944,A -85,B 0,C 180,E1 12034.436,E2 12034.436} C_VEL
LIN {X 0,Y 393.613,Z 685.126,A -85,B 0,C 180,E1 12031.886,E2 12031.886} C_VEL
LIN {X 0,Y 400.624,Z 699.139,A -85,B 0,C 180,E1 12029.268,E2 12029.268} C_VEL
LIN {X 0,Y 402.59,Z 703.512,A -85,B 0,C 180,E1 12028.573,E2 12028.573} C_VEL
LIN {X 0,Y 404.22,Z 734.044,A -85,B 0,C 180,E1 12027.096,E2 12027.096} C_VEL
LIN {X 0,Y 389.755,Z 945.325,A -85,B 0,C 180,E1 12023.637,E2 12023.637} C_VEL
LIN {X 0,Y 386.747,Z 968.366,A -85,B 0,C 180,E1 12023.106,E2 12023.106} C_VEL
LIN {X 0,Y 382.613,Z 990.681,A -85,B 0,C 180,E1 12022.416,E2 12022.416} C_VEL
LIN {X 0,Y 377.794,Z 1010.929,A -85,B 0,C 180,E1 12021.571,E2 12021.571} C_VEL
LIN {X 0,Y 371.656,Z 1032.566,A -85,B 0,C 180,E1 12020.422,E2 12020.422} C_VEL
LIN {X 0,Y 365.18,Z 1052.015,A -85,B 0,C 180,E1 12019.125,E2 12019.125} C_VEL
LIN {X 0,Y 357.537,Z 1072.059,A -85,B 0,C 180,E1 12017.466,E2 12017.466} C_VEL
LIN {X 0,Y 349.764,Z 1090.404,A -85,B 0,C 180,E1 12015.616,E2 12015.616} C_VEL
LIN {X 0,Y 341.581,Z 1107.713,A -85,B 0,C 180,E1 12013.462,E2 12013.462} C_VEL
LIN {X 0,Y 332.938,Z 1124.674,A -85,B 0,C 180,E1 12010.895,E2 12010.895} C_VEL
LIN {X 0,Y 324.996,Z 1139.315,A -85,B 0,C 180,E1 12008.198,E2 12008.198} C_VEL
LIN {X 0,Y 317.391,Z 1152.599,A -85,B 0,C 180,E1 12005.204,E2 12005.204} C_VEL
LIN {X 0,Y 310.317,Z 1164.76,A -85,B 0,C 180,E1 12001.898,E2 12001.898} C_VEL
LIN {X 0,Y 303.95,Z 1175.457,A -85,B 0,C 180,E1 11998.274,E2 11998.274} C_VEL
LIN {X 0,Y 298.271,Z 1185.303,A -85,B 0,C 180,E1 11994.14,E2 11994.14} C_VEL
LIN {X 0,Y 294.13,Z 1192.93,A -85,B 0,C 180,E1 11990.08,E2 11990.08} C_VEL
LIN {X 0,Y 291.086,Z 1199.153,A -85,B 0,C 180,E1 11985.745,E2 11985.745} C_VEL
LIN {X 0,Y 289.236,Z 1203.852,A -85,B 0,C 180,E1 11981.364,E2 11981.364} C_VEL
LIN {X 0,Y 288.324,Z 1206.855,A -85,B 0,C 180,E1 11976.971,E2 11976.971} C_VEL
LIN {X 0,Y 288.043,Z 1208.508,A -85,B 0,C 180,E1 11972.586,E2 11972.586} C_VEL
LIN {X 0,Y 288.017,Z 1208.649,A -85,B 0,C 180,E1 11968.608,E2 11968.608} C_VEL
LIN {X 0,Y 288.163,Z 1207.697,A -85,B 0,C 180,E1 11964.624,E2 11964.624} C_VEL
LIN {X 0,Y 288.788,Z 1205.17,A -85,B 0,C 180,E1 11960.233,E2 11960.233} C_VEL
LIN {X 0,Y 290.252,Z 1201.223,A -85,B 0,C 180,E1 11955.843,E2 11955.843} C_VEL
LIN {X 0,Y 292.82,Z 1195.55,A -85,B 0,C 180,E1 11951.485,E2 11951.485} C_VEL
LIN {X 0,Y 296.674,Z 1188.281,A -85,B 0,C 180,E1 11947.196,E2 11947.196} C_VEL
LIN {X 0,Y 301.618,Z 1179.56,A -85,B 0,C 180,E1 11943.203,E2 11943.203} C_VEL
LIN {X 0,Y 307.829,Z 1168.996,A -85,B 0,C 180,E1 11939.34,E2 11939.34} C_VEL
LIN {X 0,Y 314.914,Z 1157.102,A -85,B 0,C 180,E1 11935.807,E2 11935.807} C_VEL
LIN {X 0,Y 322.639,Z 1143.635,A -85,B 0,C 180,E1 11932.598,E2 11932.598} C_VEL
LIN {X 0,Y 331.31,Z 1127.94,A -85,B 0,C 180,E1 11929.545,E2 11929.545} C_VEL
LIN {X 0,Y 339.575,Z 1112.129,A -85,B 0,C 180,E1 11927.028,E2 11927.028} C_VEL
LIN {X 0,Y 347.617,Z 1095.308,A -85,B 0,C 180,E1 11924.846,E2 11924.846} C_VEL
LIN {X 0,Y 355.593,Z 1077.27,A -85,B 0,C 180,E1 11922.906,E2 11922.906} C_VEL
LIN {X 0,Y 362.866,Z 1058.773,A -85,B 0,C 180,E1 11921.284,E2 11921.284} C_VEL
LIN {X 0,Y 370.181,Z 1037.719,A -85,B 0,C 180,E1 11919.787,E2 11919.787} C_VEL
LIN {X 0,Y 376.282,Z 1017.404,A -85,B 0,C 180,E1 11918.628,E2 11918.628} C_VEL
LIN {X 0,Y 381.554,Z 996.107,A -85,B 0,C 180,E1 11917.685,E2 11917.685} C_VEL
LIN {X 0,Y 386.004,Z 974.104,A -85,B 0,C 180,E1 11916.941,E2 11916.941} C_VEL
LIN {X 0,Y 389.206,Z 951.994,A -85,B 0,C 180,E1 11916.395,E2 11916.395} C_VEL
LIN {X 0,Y 391.68,Z 921.959,A -85,B 0,C 180,E1 11915.848,E2 11915.848} C_VEL
LIN {X 0,Y 397.565,Z 833.257,A -85,B 0,C 180,E1 11914.398,E2 11914.398} C_VEL
LIN {X 0,Y 397.574,Z 825.679,A -85,B 0,C 180,E1 11914.155,E2 11914.155} C_VEL
LIN {X 0,Y 395.76,Z 805.931,A -85,B 0,C 180,E1 11913.052,E2 11913.052} C_VEL
LIN {X 0,Y 395.835,Z 799.418,A -85,B 0,C 180,E1 11912.849,E2 11912.849} C_VEL
LIN {X 0,Y 400.448,Z 733.909,A -85,B 0,C 180,E1 11911.772,E2 11911.772} C_VEL
LIN {X 0,Y 399.031,Z 707.901,A -85,B 0,C 180,E1 11910.451,E2 11910.451} C_VEL
LIN {X 0,Y 392.03,Z 693.483,A -85,B 0,C 180,E1 11907.778,E2 11907.778} C_VEL
LIN {X 0,Y 385.996,Z 681.939,A -85,B 0,C 180,E1 11905.181,E2 11905.181} C_VEL
LIN {X 0,Y 381.499,Z 673.669,A -85,B 0,C 180,E1 11902.987,E2 11902.987} C_VEL
LIN {X 0,Y 377.217,Z 665.916,A -85,B 0,C 180,E1 11900.603,E2 11900.603} C_VEL
LIN {X 0,Y 373.489,Z 659.368,A -85,B 0,C 180,E1 11898.173,E2 11898.173} C_VEL
LIN {X 0,Y 369.58,Z 652.55,A -85,B 0,C 180,E1 11895.054,E2 11895.054} C_VEL
LIN {X 0,Y 367.802,Z 649.501,A -85,B 0,C 180,E1 11893.293,E2 11893.293} C_VEL
LIN {X 0,Y 365.89,Z 645.904,A -85,B 0,C 180,E1 11890.869,E2 11890.869} C_VEL
LIN {X 0,Y 363.971,Z 641.79,A -85,B 0,C 180,E1 11886.943,E2 11886.943} C_VEL
LIN {X 0,Y 363.581,Z 640.119,A -85,B 0,C 180,E1 11881.891,E2 11881.891} C_VEL
LIN {X 0,Y 364.925,Z 640.622,A -85,B 0,C 180,E1 11878.116,E2 11878.116} C_VEL
LIN {X 0,Y 368.846,Z 644.057,A -85,B 0,C 180,E1 11873.15,E2 11873.15} C_VEL
LIN {X 0,Y 373.324,Z 649.446,A -85,B 0,C 180,E1 11869.428,E2 11869.428} C_VEL
LIN {X 0,Y 377.442,Z 654.618,A -85,B 0,C 180,E1 11866.753,E2 11866.753} C_VEL
LIN {X 0,Y 383.086,Z 662.017,A -85,B 0,C 180,E1 11863.705,E2 11863.705} C_VEL
LIN {X 0,Y 389.541,Z 671.311,A -85,B 0,C 180,E1 11860.741,E2 11860.741} C_VEL
LIN {X 0,Y 396.683,Z 682.276,A -85,B 0,C 180,E1 11857.901,E2 11857.901} C_VEL
LIN {X 0,Y 403.717,Z 694.053,A -85,B 0,C 180,E1 11855.412,E2 11855.412} C_VEL
LIN {X 0,Y 404.923,Z 696.426,A -85,B 0,C 180,E1 11855,E2 11855} C_VEL
LIN {X 0,Y 386.591,Z 927.484,A -85,B 0,C 180,E1 11850.943,E2 11850.943} C_VEL
LIN {X 0,Y 383.348,Z 952.783,A -85,B 0,C 180,E1 11850.335,E2 11850.335} C_VEL
LIN {X 0,Y 379.649,Z 973.599,A -85,B 0,C 180,E1 11849.656,E2 11849.656} C_VEL
LIN {X 0,Y 374.317,Z 997.442,A -85,B 0,C 180,E1 11848.653,E2 11848.653} C_VEL
LIN {X 0,Y 368.911,Z 1017.482,A -85,B 0,C 180,E1 11847.592,E2 11847.592} C_VEL
LIN {X 0,Y 361.553,Z 1040.868,A -85,B 0,C 180,E1 11846.061,E2 11846.061} C_VEL
LIN {X 0,Y 354.368,Z 1060.872,A -85,B 0,C 180,E1 11844.461,E2 11844.461} C_VEL
LIN {X 0,Y 346.401,Z 1080.654,A -85,B 0,C 180,E1 11842.539,E2 11842.539} C_VEL
LIN {X 0,Y 338.479,Z 1098.728,A -85,B 0,C 180,E1 11840.442,E2 11840.442} C_VEL
LIN {X 0,Y 329.699,Z 1117.163,A -85,B 0,C 180,E1 11837.857,E2 11837.857} C_VEL
LIN {X 0,Y 321.344,Z 1133.838,A -85,B 0,C 180,E1 11835.063,E2 11835.063} C_VEL
LIN {X 0,Y 313.045,Z 1149.462,A -85,B 0,C 180,E1 11831.877,E2 11831.877} C_VEL
LIN {X 0,Y 305.501,Z 1163.562,A -85,B 0,C 180,E1 11828.451,E2 11828.451} C_VEL
LIN {X 0,Y 298.632,Z 1176.208,A -85,B 0,C 180,E1 11824.693,E2 11824.693} C_VEL
LIN {X 0,Y 292.566,Z 1187.845,A -85,B 0,C 180,E1 11820.542,E2 11820.542} C_VEL
LIN {X 0,Y 287.849,Z 1197.386,A -85,B 0,C 180,E1 11816.336,E2 11816.336} C_VEL
LIN {X 0,Y 284.125,Z 1205.968,A -85,B 0,C 180,E1 11811.685,E2 11811.685} C_VEL
LIN {X 0,Y 281.858,Z 1212.217,A -85,B 0,C 180,E1 11807.336,E2 11807.336} C_VEL
LIN {X 0,Y 280.523,Z 1217.334,A -85,B 0,C 180,E1 11802.767,E2 11802.767} C_VEL
LIN {X 0,Y 280.027,Z 1220.621,A -85,B 0,C 180,E1 11798.418,E2 11798.418} C_VEL
LIN {X 0,Y 279.956,Z 1222.4,A -85,B 0,C 180,E1 11794.712,E2 11794.712} C_VEL
LIN {X 0,Y 279.983,Z 1223.192,A -85,B 0,C 180,E1 11791.023,E2 11791.023} C_VEL
LIN {X 0,Y 279.961,Z 1222.894,A -85,B 0,C 180,E1 11786.724,E2 11786.724} C_VEL
LIN {X 0,Y 279.982,Z 1221.204,A -85,B 0,C 180,E1 11782.614,E2 11782.614} C_VEL
LIN {X 0,Y 280.286,Z 1218.499,A -85,B 0,C 180,E1 11778.685,E2 11778.685} C_VEL
LIN {X 0,Y 281.326,Z 1214.035,A -85,B 0,C 180,E1 11774.118,E2 11774.118} C_VEL
LIN {X 0,Y 283.363,Z 1207.819,A -85,B 0,C 180,E1 11769.554,E2 11769.554} C_VEL
LIN {X 0,Y 286.611,Z 1200.115,A -85,B 0,C 180,E1 11765.032,E2 11765.032} C_VEL
LIN {X 0,Y 291.161,Z 1190.482,A -85,B 0,C 180,E1 11760.589,E2 11760.589} C_VEL
LIN {X 0,Y 296.785,Z 1179.665,A -85,B 0,C 180,E1 11756.461,E2 11756.461} C_VEL
LIN {X 0,Y 303.498,Z 1167.03,A -85,B 0,C 180,E1 11752.56,E2 11752.56} C_VEL
LIN {X 0,Y 310.953,Z 1153.275,A -85,B 0,C 180,E1 11749.008,E2 11749.008} C_VEL
LIN {X 0,Y 318.751,Z 1138.485,A -85,B 0,C 180,E1 11745.864,E2 11745.864} C_VEL
LIN {X 0,Y 327.396,Z 1121.63,A -85,B 0,C 180,E1 11742.866,E2 11742.866} C_VEL
LIN {X 0,Y 335.441,Z 1104.944,A -85,B 0,C 180,E1 11740.405,E2 11740.405} C_VEL
LIN {X 0,Y 344.217,Z 1085.489,A -85,B 0,C 180,E1 11738.012,E2 11738.012} C_VEL
LIN {X 0,Y 351.7,Z 1067.339,A -85,B 0,C 180,E1 11736.158,E2 11736.158} C_VEL
LIN {X 0,Y 359.649,Z 1045.97,A -85,B 0,C 180,E1 11734.342,E2 11734.342} C_VEL
LIN {X 0,Y 365.984,Z 1026.732,A -85,B 0,C 180,E1 11732.995,E2 11732.995} C_VEL
LIN {X 0,Y 372.481,Z 1003.956,A -85,B 0,C 180,E1 11731.687,E2 11731.687} C_VEL
LIN {X 0,Y 377.45,Z 983.179,A -85,B 0,C 180,E1 11730.729,E2 11730.729} C_VEL
LIN {X 0,Y 382.262,Z 958.237,A -85,B 0,C 180,E1 11729.841,E2 11729.841} C_VEL
LIN {X 0,Y 385.591,Z 935.229,A -85,B 0,C 180,E1 11729.233,E2 11729.233} C_VEL
LIN {X 0,Y 388.819,Z 898.42,A -85,B 0,C 180,E1 11728.539,E2 11728.539} C_VEL
LIN {X 0,Y 404.778,Z 695.985,A -85,B 0,C 180,E1 11725.006,E2 11725.006} C_VEL
LIN {X 0,Y 397.669,Z 684.043,A -85,B 0,C 180,E1 11722.547,E2 11722.547} C_VEL
LIN {X 0,Y 390.984,Z 673.572,A -85,B 0,C 180,E1 11719.963,E2 11719.963} C_VEL
LIN {X 0,Y 384.606,Z 664.358,A -85,B 0,C 180,E1 11717.162,E2 11717.162} C_VEL
LIN {X 0,Y 379.371,Z 657.171,A -85,B 0,C 180,E1 11714.5,E2 11714.5} C_VEL
LIN {X 0,Y 375.5,Z 652.224,A -85,B 0,C 180,E1 11712.222,E2 11712.222} C_VEL
LIN {X 0,Y 372.133,Z 648.041,A -85,B 0,C 180,E1 11709.902,E2 11709.902} C_VEL
LIN {X 0,Y 368.096,Z 643.293,A -85,B 0,C 180,E1 11706.394,E2 11706.394} C_VEL
LIN {X 0,Y 364.394,Z 640.102,A -85,B 0,C 180,E1 11701.415,E2 11701.415} C_VEL
LIN {X 0,Y 363.242,Z 639.716,A -85,B 0,C 180,E1 11697.949,E2 11697.949} C_VEL
LIN {X 0,Y 363.764,Z 641.707,A -85,B 0,C 180,E1 11692.577,E2 11692.577} C_VEL
LIN {X 0,Y 366.179,Z 646.745,A -85,B 0,C 180,E1 11688.182,E2 11688.182} C_VEL
LIN {X 0,Y 369.035,Z 651.798,A -85,B 0,C 180,E1 11685.084,E2 11685.084} C_VEL
LIN {X 0,Y 371.751,Z 656.686,A -85,B 0,C 180,E1 11682.79,E2 11682.79} C_VEL
LIN {X 0,Y 375.686,Z 663.456,A -85,B 0,C 180,E1 11680.082,E2 11680.082} C_VEL
LIN {X 0,Y 380.564,Z 672.083,A -85,B 0,C 180,E1 11677.28,E2 11677.28} C_VEL
LIN {X 0,Y 385.536,Z 681.282,A -85,B 0,C 180,E1 11674.828,E2 11674.828} C_VEL
LIN {X 0,Y 391.222,Z 692.077,A -85,B 0,C 180,E1 11672.362,E2 11672.362} C_VEL
LIN {X 0,Y 397.849,Z 705.671,A -85,B 0,C 180,E1 11669.804,E2 11669.804} C_VEL
LIN {X 0,Y 398.941,Z 708.335,A -85,B 0,C 180,E1 11669.396,E2 11669.396} C_VEL
LIN {X 0,Y 400.208,Z 735.615,A -85,B 0,C 180,E1 11668.069,E2 11668.069} C_VEL
LIN {X 0,Y 385.423,Z 945.06,A -85,B 0,C 180,E1 11664.636,E2 11664.636} C_VEL
LIN {X 0,Y 382.344,Z 968.138,A -85,B 0,C 180,E1 11664.106,E2 11664.106} C_VEL
LIN {X 0,Y 378.166,Z 990.26,A -85,B 0,C 180,E1 11663.427,E2 11663.427} C_VEL
LIN {X 0,Y 373.239,Z 1010.538,A -85,B 0,C 180,E1 11662.588,E2 11662.588} C_VEL
LIN {X 0,Y 366.957,Z 1032.228,A -85,B 0,C 180,E1 11661.444,E2 11661.444} C_VEL
LIN {X 0,Y 360.528,Z 1051.11,A -85,B 0,C 180,E1 11660.193,E2 11660.193} C_VEL
LIN {X 0,Y 352.779,Z 1071.069,A -85,B 0,C 180,E1 11658.56,E2 11658.56} C_VEL
LIN {X 0,Y 344.773,Z 1089.541,A -85,B 0,C 180,E1 11656.711,E2 11656.711} C_VEL
LIN {X 0,Y 336.327,Z 1106.976,A -85,B 0,C 180,E1 11654.555,E2 11654.555} C_VEL
LIN {X 0,Y 327.902,Z 1123.164,A -85,B 0,C 180,E1 11652.132,E2 11652.132} C_VEL
LIN {X 0,Y 320.074,Z 1137.122,A -85,B 0,C 180,E1 11649.588,E2 11649.588} C_VEL
LIN {X 0,Y 311.218,Z 1152.172,A -85,B 0,C 180,E1 11646.238,E2 11646.238} C_VEL
LIN {X 0,Y 303.825,Z 1164.404,A -85,B 0,C 180,E1 11642.888,E2 11642.888} C_VEL
LIN {X 0,Y 297.127,Z 1175.187,A -85,B 0,C 180,E1 11639.205,E2 11639.205} C_VEL
LIN {X 0,Y 291.363,Z 1184.743,A -85,B 0,C 180,E1 11635.184,E2 11635.184} C_VEL
LIN {X 0,Y 286.887,Z 1192.469,A -85,B 0,C 180,E1 11631.037,E2 11631.037} C_VEL
LIN {X 0,Y 283.368,Z 1199.227,A -85,B 0,C 180,E1 11626.305,E2 11626.305} C_VEL
LIN {X 0,Y 281.328,Z 1204.061,A -85,B 0,C 180,E1 11621.688,E2 11621.688} C_VEL
LIN {X 0,Y 280.35,Z 1207.061,A -85,B 0,C 180,E1 11617.171,E2 11617.171} C_VEL
LIN {X 0,Y 280.047,Z 1208.713,A -85,B 0,C 180,E1 11612.66,E2 11612.66} C_VEL
LIN {X 0,Y 280.02,Z 1208.853,A -85,B 0,C 180,E1 11608.568,E2 11608.568} C_VEL
LIN {X 0,Y 280.178,Z 1207.901,A -85,B 0,C 180,E1 11604.471,E2 11604.471} C_VEL
LIN {X 0,Y 280.857,Z 1205.377,A -85,B 0,C 180,E1 11599.954,E2 11599.954} C_VEL
LIN {X 0,Y 282.414,Z 1201.43,A -85,B 0,C 180,E1 11595.442,E2 11595.442} C_VEL
LIN {X 0,Y 285.143,Z 1195.761,A -85,B 0,C 180,E1 11590.967,E2 11590.967} C_VEL
LIN {X 0,Y 289.208,Z 1188.5,A -85,B 0,C 180,E1 11586.573,E2 11586.573} C_VEL
LIN {X 0,Y 294.393,Z 1179.784,A -85,B 0,C 180,E1 11582.49,E2 11582.49} C_VEL
LIN {X 0,Y 300.875,Z 1169.233,A -85,B 0,C 180,E1 11578.551,E2 11578.551} C_VEL
LIN {X 0,Y 308.245,Z 1157.35,A -85,B 0,C 180,E1 11574.961,E2 11574.961} C_VEL
LIN {X 0,Y 316.248,Z 1143.899,A -85,B 0,C 180,E1 11571.707,E2 11571.707} C_VEL
LIN {X 0,Y 325.336,Z 1128.009,A -85,B 0,C 180,E1 11568.583,E2 11568.583} C_VEL
LIN {X 0,Y 333.997,Z 1111.948,A -85,B 0,C 180,E1 11566.011,E2 11566.011} C_VEL
LIN {X 0,Y 342.333,Z 1094.978,A -85,B 0,C 180,E1 11563.807,E2 11563.807} C_VEL
LIN {X 0,Y 350.78,Z 1076.272,A -85,B 0,C 180,E1 11561.809,E2 11561.809} C_VEL
LIN {X 0,Y 358.129,Z 1058.016,A -85,B 0,C 180,E1 11560.219,E2 11560.219} C_VEL
LIN {X 0,Y 365.449,Z 1037.366,A -85,B 0,C 180,E1 11558.762,E2 11558.762} C_VEL
LIN {X 0,Y 371.698,Z 1017.025,A -85,B 0,C 180,E1 11557.609,E2 11557.609} C_VEL
LIN {X 0,Y 377.089,Z 995.663,A -85,B 0,C 180,E1 11556.671,E2 11556.671} C_VEL
LIN {X 0,Y 381.657,Z 973.442,A -85,B 0,C 180,E1 11555.928,E2 11555.928} C_VEL
LIN {X 0,Y 384.895,Z 951.478,A -85,B 0,C 180,E1 11555.39,E2 11555.39} C_VEL
LIN {X 0,Y 387.436,Z 921.242,A -85,B 0,C 180,E1 11554.841,E2 11554.841} C_VEL
LIN {X 0,Y 395.835,Z 799.418,A -85,B 0,C 180,E1 11552.849,E2 11552.849} C_VEL
LIN {X 0,Y 395.869,Z 791.844,A -85,B 0,C 180,E1 11552.598,E2 11552.598} C_VEL
LIN {X 0,Y 394.272,Z 772.097,A -85,B 0,C 180,E1 11551.482,E2 11551.482} C_VEL
LIN {X 0,Y 394.412,Z 765.583,A -85,B 0,C 180,E1 11551.286,E2 11551.286} C_VEL
LIN {X 0,Y 396.569,Z 735.299,A -85,B 0,C 180,E1 11550.774,E2 11550.774} C_VEL
LIN {X 0,Y 395.5,Z 712.767,A -85,B 0,C 180,E1 11549.621,E2 11549.621} C_VEL
LIN {X 0,Y 389.081,Z 699.23,A -85,B 0,C 180,E1 11547.057,E2 11547.057} C_VEL
LIN {X 0,Y 383.399,Z 688.129,A -85,B 0,C 180,E1 11544.498,E2 11544.498} C_VEL
LIN {X 0,Y 378.666,Z 679.127,A -85,B 0,C 180,E1 11542.058,E2 11542.058} C_VEL
LIN {X 0,Y 373.279,Z 669.121,A -85,B 0,C 180,E1 11538.75,E2 11538.75} C_VEL
LIN {X 0,Y 368.357,Z 660.407,A -85,B 0,C 180,E1 11534.864,E2 11534.864} C_VEL
LIN {X 0,Y 366.542,Z 657.191,A -85,B 0,C 180,E1 11533.006,E2 11533.006} C_VEL
LIN {X 0,Y 364.705,Z 653.644,A -85,B 0,C 180,E1 11530.585,E2 11530.585} C_VEL
LIN {X 0,Y 362.948,Z 649.682,A -85,B 0,C 180,E1 11526.803,E2 11526.803} C_VEL
LIN {X 0,Y 362.635,Z 648.048,A -85,B 0,C 180,E1 11521.738,E2 11521.738} C_VEL
LIN {X 0,Y 364.034,Z 648.642,A -85,B 0,C 180,E1 11517.954,E2 11517.954} C_VEL
LIN {X 0,Y 367.621,Z 651.855,A -85,B 0,C 180,E1 11513.362,E2 11513.362} C_VEL
LIN {X 0,Y 371.902,Z 657.124,A -85,B 0,C 180,E1 11509.701,E2 11509.701} C_VEL
LIN {X 0,Y 375.816,Z 662.14,A -85,B 0,C 180,E1 11507.086,E2 11507.086} C_VEL
LIN {X 0,Y 381.334,Z 669.541,A -85,B 0,C 180,E1 11504.019,E2 11504.019} C_VEL
LIN {X 0,Y 387.671,Z 678.927,A -85,B 0,C 180,E1 11501.035,E2 11501.035} C_VEL
LIN {X 0,Y 394.342,Z 689.422,A -85,B 0,C 180,E1 11498.311,E2 11498.311} C_VEL
LIN {X 0,Y 400.85,Z 700.537,A -85,B 0,C 180,E1 11495.94,E2 11495.94} C_VEL
LIN {X 0,Y 382.335,Z 928.255,A -85,B 0,C 180,E1 11491.947,E2 11491.947} C_VEL
LIN {X 0,Y 378.922,Z 953.934,A -85,B 0,C 180,E1 11491.326,E2 11491.326} C_VEL
LIN {X 0,Y 375.118,Z 974.727,A -85,B 0,C 180,E1 11490.645,E2 11490.645} C_VEL
LIN {X 0,Y 369.64,Z 998.432,A -85,B 0,C 180,E1 11489.641,E2 11489.641} C_VEL
LIN {X 0,Y 363.792,Z 1019.484,A -85,B 0,C 180,E1 11488.519,E2 11488.519} C_VEL
LIN {X 0,Y 356.684,Z 1041.284,A -85,B 0,C 180,E1 11487.079,E2 11487.079} C_VEL
LIN {X 0,Y 349.273,Z 1061.36,A -85,B 0,C 180,E1 11485.47,E2 11485.47} C_VEL
LIN {X 0,Y 340.857,Z 1081.588,A -85,B 0,C 180,E1 11483.489,E2 11483.489} C_VEL
LIN {X 0,Y 332.16,Z 1100.801,A -85,B 0,C 180,E1 11481.227,E2 11481.227} C_VEL
LIN {X 0,Y 323.413,Z 1118.382,A -85,B 0,C 180,E1 11478.699,E2 11478.699} C_VEL
LIN {X 0,Y 314.809,Z 1134.885,A -85,B 0,C 180,E1 11475.872,E2 11475.872} C_VEL
LIN {X 0,Y 306.477,Z 1149.972,A -85,B 0,C 180,E1 11472.733,E2 11472.733} C_VEL
LIN {X 0,Y 298.263,Z 1164.618,A -85,B 0,C 180,E1 11469.067,E2 11469.067} C_VEL
LIN {X 0,Y 291.51,Z 1176.555,A -85,B 0,C 180,E1 11465.426,E2 11465.426} C_VEL
LIN {X 0,Y 284.995,Z 1188.421,A -85,B 0,C 180,E1 11461.046,E2 11461.046} C_VEL
LIN {X 0,Y 280.249,Z 1197.578,A -85,B 0,C 180,E1 11456.878,E2 11456.878} C_VEL
LIN {X 0,Y 276.199,Z 1206.386,A -85,B 0,C 180,E1 11451.892,E2 11451.892} C_VEL
LIN {X 0,Y 273.954,Z 1212.27,A -85,B 0,C 180,E1 11447.633,E2 11447.633} C_VEL
LIN {X 0,Y 272.507,Z 1217.471,A -85,B 0,C 180,E1 11442.718,E2 11442.718} C_VEL
LIN {X 0,Y 272.029,Z 1220.534,A -85,B 0,C 180,E1 11438.454,E2 11438.454} C_VEL
LIN {X 0,Y 271.958,Z 1222.267,A -85,B 0,C 180,E1 11434.639,E2 11434.639} C_VEL
LIN {X 0,Y 271.984,Z 1223.044,A -85,B 0,C 180,E1 11430.55,E2 11430.55} C_VEL
LIN {X 0,Y 271.968,Z 1222.545,A -85,B 0,C 180,E1 11426.206,E2 11426.206} C_VEL
LIN {X 0,Y 271.989,Z 1220.876,A -85,B 0,C 180,E1 11422.183,E2 11422.183} C_VEL
LIN {X 0,Y 272.364,Z 1218.12,A -85,B 0,C 180,E1 11418.137,E2 11418.137} C_VEL
LIN {X 0,Y 273.617,Z 1213.293,A -85,B 0,C 180,E1 11413.221,E2 11413.221} C_VEL
LIN {X 0,Y 275.825,Z 1207.206,A -85,B 0,C 180,E1 11408.694,E2 11408.694} C_VEL
LIN {X 0,Y 279.507,Z 1199.071,A -85,B 0,C 180,E1 11403.896,E2 11403.896} C_VEL
LIN {X 0,Y 284.275,Z 1189.655,A -85,B 0,C 180,E1 11399.514,E2 11399.514} C_VEL
LIN {X 0,Y 290.53,Z 1178.228,A -85,B 0,C 180,E1 11395.16,E2 11395.16} C_VEL
LIN {X 0,Y 297.116,Z 1166.461,A -85,B 0,C 180,E1 11391.496,E2 11391.496} C_VEL
LIN {X 0,Y 305.28,Z 1151.966,A -85,B 0,C 180,E1 11387.751,E2 11387.751} C_VEL
LIN {X 0,Y 312.855,Z 1138.184,A -85,B 0,C 180,E1 11384.807,E2 11384.807} C_VEL
LIN {X 0,Y 322.082,Z 1120.767,A -85,B 0,C 180,E1 11381.704,E2 11381.704} C_VEL
LIN {X 0,Y 330.169,Z 1104.538,A -85,B 0,C 180,E1 11379.31,E2 11379.31} C_VEL
LIN {X 0,Y 339.355,Z 1084.698,A -85,B 0,C 180,E1 11376.876,E2 11376.876} C_VEL
LIN {X 0,Y 346.912,Z 1066.858,A -85,B 0,C 180,E1 11375.062,E2 11375.062} C_VEL
LIN {X 0,Y 355.083,Z 1045.368,A -85,B 0,C 180,E1 11373.248,E2 11373.248} C_VEL
LIN {X 0,Y 361.59,Z 1026.05,A -85,B 0,C 180,E1 11371.907,E2 11371.907} C_VEL
LIN {X 0,Y 368.254,Z 1003.048,A -85,B 0,C 180,E1 11370.605,E2 11370.605} C_VEL
LIN {X 0,Y 373.351,Z 982.111,A -85,B 0,C 180,E1 11369.654,E2 11369.654} C_VEL
LIN {X 0,Y 378.05,Z 957.966,A -85,B 0,C 180,E1 11368.808,E2 11368.808} C_VEL
LIN {X 0,Y 381.501,Z 934.481,A -85,B 0,C 180,E1 11368.195,E2 11368.195} C_VEL
LIN {X 0,Y 385.319,Z 890.463,A -85,B 0,C 180,E1 11367.379,E2 11367.379} C_VEL
LIN {X 0,Y 400.642,Z 700.339,A -85,B 0,C 180,E1 11364.063,E2 11364.063} C_VEL
LIN {X 0,Y 393.535,Z 688.198,A -85,B 0,C 180,E1 11361.462,E2 11361.462} C_VEL
LIN {X 0,Y 386.342,Z 676.983,A -85,B 0,C 180,E1 11358.484,E2 11358.484} C_VEL
LIN {X 0,Y 380.243,Z 668.23,A -85,B 0,C 180,E1 11355.558,E2 11355.558} C_VEL
LIN {X 0,Y 374.741,Z 660.661,A -85,B 0,C 180,E1 11352.403,E2 11352.403} C_VEL
LIN {X 0,Y 370.731,Z 655.732,A -85,B 0,C 180,E1 11349.626,E2 11349.626} C_VEL
LIN {X 0,Y 366.954,Z 651.165,A -85,B 0,C 180,E1 11346.257,E2 11346.257} C_VEL
LIN {X 0,Y 363.418,Z 648.053,A -85,B 0,C 180,E1 11341.419,E2 11341.419} C_VEL
LIN {X 0,Y 362.267,Z 647.659,A -85,B 0,C 180,E1 11337.944,E2 11337.944} C_VEL
LIN {X 0,Y 362.8,Z 649.676,A -85,B 0,C 180,E1 11332.557,E2 11332.557} C_VEL
LIN {X 0,Y 365.08,Z 654.714,A -85,B 0,C 180,E1 11328.307,E2 11328.307} C_VEL
LIN {X 0,Y 367.824,Z 659.652,A -85,B 0,C 180,E1 11325.276,E2 11325.276} C_VEL
LIN {X 0,Y 371.498,Z 666.296,A -85,B 0,C 180,E1 11322.212,E2 11322.212} C_VEL
LIN {X 0,Y 375.368,Z 673.271,A -85,B 0,C 180,E1 11319.621,E2 11319.621} C_VEL
LIN {X 0,Y 379.295,Z 680.592,A -85,B 0,C 180,E1 11317.363,E2 11317.363} C_VEL
LIN {X 0,Y 383.695,Z 688.896,A -85,B 0,C 180,E1 11315.152,E2 11315.152} C_VEL
LIN {X 0,Y 389.609,Z 700.588,A -85,B 0,C 180,E1 11312.528,E2 11312.528} C_VEL
LIN {X 0,Y 395.349,Z 712.811,A -85,B 0,C 180,E1 11310.252,E2 11310.252} C_VEL
LIN {X 0,Y 396.333,Z 737.044,A -85,B 0,C 180,E1 11309.064,E2 11309.064} C_VEL
LIN {X 0,Y 381.214,Z 944.741,A -85,B 0,C 180,E1 11305.659,E2 11305.659} C_VEL
LIN {X 0,Y 378.059,Z 967.901,A -85,B 0,C 180,E1 11305.129,E2 11305.129} C_VEL
LIN {X 0,Y 373.842,Z 989.839,A -85,B 0,C 180,E1 11304.462,E2 11304.462} C_VEL
LIN {X 0,Y 368.804,Z 1010.144,A -85,B 0,C 180,E1 11303.629,E2 11303.629} C_VEL
LIN {X 0,Y 362.718,Z 1030.891,A -85,B 0,C 180,E1 11302.551,E2 11302.551} C_VEL
LIN {X 0,Y 356.117,Z 1049.906,A -85,B 0,C 180,E1 11301.309,E2 11301.309} C_VEL
LIN {X 0,Y 347.843,Z 1070.802,A -85,B 0,C 180,E1 11299.617,E2 11299.617} C_VEL
LIN {X 0,Y 339.617,Z 1089.299,A -85,B 0,C 180,E1 11297.768,E2 11297.768} C_VEL
LIN {X 0,Y 330.921,Z 1106.777,A -85,B 0,C 180,E1 11295.608,E2 11295.608} C_VEL
LIN {X 0,Y 321.966,Z 1123.466,A -85,B 0,C 180,E1 11293.094,E2 11293.094} C_VEL
LIN {X 0,Y 313.89,Z 1137.409,A -85,B 0,C 180,E1 11290.528,E2 11290.528} C_VEL
LIN {X 0,Y 305.159,Z 1151.748,A -85,B 0,C 180,E1 11287.312,E2 11287.312} C_VEL
LIN {X 0,Y 297.424,Z 1164.035,A -85,B 0,C 180,E1 11283.921,E2 11283.921} C_VEL
LIN {X 0,Y 290.388,Z 1174.919,A -85,B 0,C 180,E1 11280.179,E2 11280.179} C_VEL
LIN {X 0,Y 284.297,Z 1184.571,A -85,B 0,C 180,E1 11276.079,E2 11276.079} C_VEL
LIN {X 0,Y 279.526,Z 1192.344,A -85,B 0,C 180,E1 11271.839,E2 11271.839} C_VEL
LIN {X 0,Y 275.661,Z 1199.333,A -85,B 0,C 180,E1 11266.868,E2 11266.868} C_VEL
LIN {X 0,Y 273.503,Z 1204.079,A -85,B 0,C 180,E1 11262.242,E2 11262.242} C_VEL
LIN {X 0,Y 272.408,Z 1207.161,A -85,B 0,C 180,E1 11257.593,E2 11257.593} C_VEL
LIN {X 0,Y 272.063,Z 1208.837,A -85,B 0,C 180,E1 11253.16,E2 11253.16} C_VEL
LIN {X 0,Y 272.021,Z 1209.078,A -85,B 0,C 180,E1 11248.736,E2 11248.736} C_VEL
LIN {X 0,Y 272.17,Z 1208.201,A -85,B 0,C 180,E1 11244.622,E2 11244.622} C_VEL
LIN {X 0,Y 272.927,Z 1205.582,A -85,B 0,C 180,E1 11239.659,E2 11239.659} C_VEL
LIN {X 0,Y 274.591,Z 1201.637,A -85,B 0,C 180,E1 11235.017,E2 11235.017} C_VEL
LIN {X 0,Y 277.49,Z 1195.974,A -85,B 0,C 180,E1 11230.421,E2 11230.421} C_VEL
LIN {X 0,Y 281.778,Z 1188.719,A -85,B 0,C 180,E1 11225.917,E2 11225.917} C_VEL
LIN {X 0,Y 287.234,Z 1179.977,A -85,B 0,C 180,E1 11221.73,E2 11221.73} C_VEL
LIN {X 0,Y 294.335,Z 1168.911,A -85,B 0,C 180,E1 11217.539,E2 11217.539} C_VEL
LIN {X 0,Y 302.059,Z 1156.936,A -85,B 0,C 180,E1 11213.9,E2 11213.9} C_VEL
LIN {X 0,Y 310.24,Z 1143.672,A -85,B 0,C 180,E1 11210.67,E2 11210.67} C_VEL
LIN {X 0,Y 319.201,Z 1128.534,A -85,B 0,C 180,E1 11207.665,E2 11207.665} C_VEL
LIN {X 0,Y 327.939,Z 1112.822,A -85,B 0,C 180,E1 11205.119,E2 11205.119} C_VEL
LIN {X 0,Y 336.726,Z 1095.544,A -85,B 0,C 180,E1 11202.844,E2 11202.844} C_VEL
LIN {X 0,Y 345.185,Z 1077.448,A -85,B 0,C 180,E1 11200.887,E2 11200.887} C_VEL
LIN {X 0,Y 353.017,Z 1058.517,A -85,B 0,C 180,E1 11199.228,E2 11199.228} C_VEL
LIN {X 0,Y 360.839,Z 1037.014,A -85,B 0,C 180,E1 11197.712,E2 11197.712} C_VEL
LIN {X 0,Y 367.234,Z 1016.646,A -85,B 0,C 180,E1 11196.565,E2 11196.565} C_VEL
LIN {X 0,Y 372.745,Z 995.224,A -85,B 0,C 180,E1 11195.633,E2 11195.633} C_VEL
LIN {X 0,Y 377.454,Z 972.651,A -85,B 0,C 180,E1 11194.889,E2 11194.889} C_VEL
LIN {X 0,Y 380.726,Z 950.805,A -85,B 0,C 180,E1 11194.358,E2 11194.358} C_VEL
LIN {X 0,Y 383.353,Z 920.047,A -85,B 0,C 180,E1 11193.803,E2 11193.803} C_VEL
LIN {X 0,Y 394.412,Z 765.583,A -85,B 0,C 180,E1 11191.286,E2 11191.286} C_VEL
LIN {X 0,Y 394.601,Z 757.977,A -85,B 0,C 180,E1 11191.06,E2 11191.06} C_VEL
LIN {X 0,Y 393.83,Z 746.523,A -85,B 0,C 180,E1 11190.422,E2 11190.422} C_VEL
LIN {X 0,Y 392.625,Z 732.027,A -85,B 0,C 180,E1 11189.521,E2 11189.521} C_VEL
LIN {X 0,Y 391.968,Z 717.415,A -85,B 0,C 180,E1 11188.741,E2 11188.741} C_VEL
